FUNCTION_BLOCK "STD_LineSecStdSub2"	// FB 90
TITLE = Line and section control standard subroutines
//COPYRIGHT:   (C) 2004 BY  BUHLER LTD.
//                          CH-9240 UZWIL  SWITZERLAND
//
//PRODUCT:      STD_MU664    
//
//TITLE:        Line and section control standard subroutines
//              
//              Standardfunktionen für Linien und Sektionen              
//              
//
//--------------------------------------------------------------------------------
//
//IDENT:        AUTOR:              DEPT:                              DATE:
//STD_FB90.4.2  Ph. Engler          MU664                              27-Oct-2005
//              Sub2001: CmdStepOff modifyed
//STD_FB90.4.1  Ph. Engler          MU664                              22-Oct-2004
//              Sub2002: Extended section commands
//STD_FB90.4.0  Ph. Engler          MU664                              02-Sep-2004
//              Sub1055: StaDPFault as SubCode
//              Sub2055: StaDPFault as SubCode
//STD_FB90.3.4  Ph. Engler          MU664                              02-Jul-2004
//              Sub2003: No immediate stop anymore, its done from FC60 Move data
//STD_FB90.3.3  Ph. Engler          MU664                              23-Jun-2004
//              Sub1061/1062: BEA added
//STD_FB90.3.2  Ph. Engler          MU664                              02-Apr-2004
//              Sub2071: SectionState integrated   
//STD_FB90.3.1  Ph. Engler          MU664                              25-Mar-2004
//              Sub1061: Fault corrected, wrong tmp
//STD_FB90.3.0  Ph. Engler          MU664                              19-Feb-2004
//              Sub1061: General group info code for 64 objects
//STD_FB90.2.6  Ph. Engler          MU664                              12-Feb-2004
//              Sub1062: Maintenance info code
//STD_FB90.2.5  Ph. Engler          MU664                              28-Aug-2003
//              Sub1055: Handling of feeding section
//STD_FB90.2.4  Ph. Engler          MU664                              04-Aug-2003
//              Sub1061: Use LC to handle tmpLin_GenGrpCoulorCode
//STD_FB90.2.3  Ph. Engler          MU664                              29-Jul-2003
//              Sub1061: InOutValue3 stored to tmpDInt
//STD_FB90.2.2  Ph. Engler          MU664                              21-Jun-2003
//              Sub1051 corrected, yellow and blue
//STD_FB90.2.1  A.Egli              CT3                                14-Mai-2003
//              Sub1001: On Off Command Line
//STD_FB90.2.0  A.Egli              CT3                                18-Oct-2002
//              New release: Function moved from FC120 to FB90
//STD_FC120.1.12Ph. Engler          MU664                              23-Aug-2002
//              - Function (4,1) added: Search group manual mode
//STD_FC120.1.11Ph. Engler          MU664                              30-Apr-2002
//              - Function (1,55) and (2,55) modified: Stopping/Stopped
//STD_FC120.1.10Ph. Engler          MU664                              21-Mar-2002
//              - Function (2,55): starting until S.ToSSW.infStarted
//STD_FC120.1.9 Ph. Engler          MU664                              12-Mar-2002
//              Status codes for WinCoS implemented:
//              - General group colour code
//              - Line and Section info code
//STD_FC120.1.8 Ph. Engler          MU664                              20-Mar-2001
//              Line status colour for 2-4 section implemented
//STD_FC120.1.7 Ph. Engler          MU664                              20-Dec-2000
//              Pre stop weight for cmdSequenceStop
//STD_FC120.1.6 Ph. Engler          MU664                              14-Dec-2000
//              - Substitude Bincode into recipe extended, InCode 3 
//              - JS Job paramter flags (2,2) Sta-Address corrected
//STD_FC120.1.5 Ph. Engler          MU664                              01-Nov-2000
//              CmdSequenceStop only if section is in StActive           
//STD_FC120.1.4 Ph. Engler          MU664                              19-Okt-2000
//              Update SND-Binlist staSameSndRcv:
//               Suppression of the error meassage 'bin not found'
//STD_FC120.1.3 Ph. Engler          MU664                              28-Jun-2000
//              Section text and colour code extension 
//              with code 702, 703 and 1402
//STD_FC120.1.2 Ph. Engler          MU664                              04-May-2000
//              LS Line state/fault protocolling (1,10)
//               esXXX corrected 
//STD_FC120.1.1 Ph. Engler          MU664                              29-Mar-2000
//              Line log messages implemented
//STD_FC120.1.0 Ph. Engler          MU664                              05-Jan-2000
//              1st Release
//
//--------------------------------------------------------------------------------
//
//PURPOSE:      
//
//RESTRICTIONS:
//
//--------------------------------------------------------------------------------
//
AUTHOR : PE
FAMILY : STD
VERSION : 4.1
VAR_INPUT
  InCode : INT ;
END_VAR
VAR
  Para : STRUCT
   ParSecNr : INT  := 1;
   ParLineDB_ParFirstSecDB : INT  := 320;
   spare4 : INT ;
   ParNextSecDB : INT ;	//Next section DB of this project line
   ParSecDataFirstByte : INT  := 240;
   ParSecDataLenNomValue : INT  := 20;
   ParSecDataLenAcValue : INT  := 20;
   ParBinDataFirstByte : INT  := 300;
   ParBinDataLength : INT  := 72;
  END_STRUCT ;
  VarTemp : STRUCT
   InOutValue1 : INT ;
   InOutValue2 : INT ;
   InOutValue3 : DINT ;
   InOutValue4 : DINT ;
   InOutValue5 : DINT ;
   InOutValue6 : DINT ;
  END_STRUCT ;
  ChangeBit : STRUCT
   spare : BYTE ;
   CBit1 : BOOL ;
   CBit2 : BOOL ;
   CBit3 : BOOL ;
   CBit4 : BOOL ;
  END_STRUCT ;
  ToASW : STRUCT
   spare00 : WORD ;
   CmdModify : BOOL ;
   CmdNewBatch : BOOL ;
   CmdDataMoved : BOOL ;
   InfSameJobPrevSec : BOOL ;
   InfSameJobNextSec : BOOL ;
   InfSameBatchPrevSec : BOOL ;
   InfSameBatchNextSec : BOOL ;
   InfSameJobLineDB : BOOL ;	//Job in reveive box is equal
   InfEmptyingTimeEnd : BOOL ;
   InfWayAdjustTimeEnd : BOOL ;
   spare32 : BOOL ;
   spare33 : BOOL ;
   spare34 : BOOL ;
   spare35 : BOOL ;
   spare36 : BOOL ;
   InfDataReady : BOOL ;
   Func : UDT 10601;
   Transition : STRUCT
    spare00 : BYTE ;
    ToPassive : BOOL ;
    ToWait : BOOL ;
    ToActive : BOOL ;
    ToReady : BOOL ;
    ToEmptying : BOOL ;
    ToEmptied : BOOL ;
    ToIdling : BOOL ;
   END_STRUCT ;
   spare10 : WORD ;
   spare12 : DWORD ;
   spare16 : DWORD ;
  END_STRUCT ;
  ToSSW : STRUCT
   InfStopped : BOOL ;
   spare01 : BOOL ;
   InfStarted : BOOL ;
   spare03 : BOOL ;
   spare04 : BOOL ;
   InfFeeding : BOOL ;
   spare06 : BOOL ;
   spare07 : BOOL ;
   spare00 : BOOL ;
   CmdGotoActive : BOOL ;
   CmdGotoReady : BOOL ;
   CmdGotoEmptying : BOOL ;
   CmdGotoEmptied : BOOL ;
   CmdGotoIdling : BOOL ;
   CmdGotoPassive : BOOL ;
   spare17 : BOOL ;
   InfReadyForNewBatch : BOOL ;
   CmdSendResult : BOOL ;
   InfPulseTimer : BOOL ;
   CmdNewWay : BOOL ;
   spare24 : BOOL ;
   spare25 : BOOL ;
   spare26 : BOOL ;
   InfReleaseEmptyingTime : BOOL ;
   Func : UDT 10601;
   InPrevSecDB : INT ;	//Previouse section DB in product flow
   InNextSecDB : INT ;	//Next section DB in product flow
   spare12 : DWORD ;
   spare16 : DWORD ;
  END_STRUCT ;
  PCWrite : STRUCT 	//PC Write : Section Data
   Hsk : STRUCT
    Q_Status : BOOL ;
    Q_Result : BOOL ;
    spare02 : BOOL ;
    spare03 : BOOL ;
    spare04 : BOOL ;
    spare05 : BOOL ;
    Q_MDEEData : BOOL ;	//Acknowledge data sended to MDEE by PCC
    Q_MYRAData : BOOL ;	//Acknowledge data sended to MYRA by PCC
    F_Define : BOOL ;
   END_STRUCT ;
   spare2 : WORD ;
   Func : UDT 10601;
   Value1 : INT ;
   Value2 : INT ;
   Value3 : INT ;
   ParWayAdjustTime : INT  := 2;
   Value5 : INT ;
   ParEmptyingTime : INT  := 20;
  END_STRUCT ;
  PCRead : STRUCT 	//PC Read : Section Data
   Hsk : STRUCT
    F_Status : BOOL ;
    F_Result : BOOL ;
    F_2 : BOOL ;
    F_3 : BOOL ;
    F_4 : BOOL ;
    F_5 : BOOL ;
    F_MDEEData : BOOL ;	//Request PCC to send data to MDEE
    F_MYRAData : BOOL ;	//Request PCC to send data to MYRA
   END_STRUCT ;
   ErrElement : INT ;
   ErrCode : INT ;
   ErrObject : INT ;	//(*new*)
   Step : STRUCT
    spare : BYTE ;
    StPassive : BOOL ;
    StWait : BOOL ;
    StActive : BOOL ;
    StReady : BOOL ;	//Line= Idling
    StEmptying : BOOL ;
    StEmptied : BOOL ;
    StIdling : BOOL ;
   END_STRUCT ;
   State : STRUCT
    spare : BYTE ;
    StStopped : BOOL ;
    StStarting : BOOL ;
    StStarted : BOOL ;
    StStopping : BOOL ;
    spare04 : BOOL ;
    StFeeding : BOOL ;
   END_STRUCT ;
   Fault : UDT 10602;
   Status : UDT 10603;
   InfoCode : INT ;
   SectionState : INT ;	//Line: GenGrpColorCode
   ExtStatus : INT ;
   OutWayAdjustTime_ExtOn : INT ;
   OutStartWarningTime : INT ;	//Copy of Startwarning modul
   OutEmptyingTime : INT ;
   Value7 : INT ;
   Value8 : INT ;
   Value9 : INT ;
   Value10 : INT ;
   Value11 : INT ;
   Value12 : INT ;
   Value13 : INT ;
   Value14 : INT ;
   Value15 : INT ;
   Value16 : INT ;
   Value17 : INT ;
   ExtFuncOn : INT ;
   Value19 : INT ;
  END_STRUCT ;
  JobNom : STRUCT 	//PC Read: Job header: Nominal values
   JobNr : DINT ;
   JobWeight : DINT ;	//Total Job weight
   BatchNo : INT  := 10;	//Number of batch requested form PC
   ScaleUsed : ARRAY  [1 .. 64 ] OF BOOL ;
   RecipeNr : INT ;
   BatchWeight : DINT ;
   BatchMinPpm : INT ;	//Minimum batch size [0.1%]
   BatchMaxPpm : INT ;	//Maximum batch size [0.1%]
   BatchNoOffset : INT ;	//Batch number of first batch
   MixingTime : INT ;	//Mixing time
   JobChangeTime : INT ;	//Job change time
   FeedingTime : INT ;	//Feeding Time
   Value13 : INT ;
   Value14 : INT ;
  END_STRUCT ;
  JobAc : STRUCT 	//PC Read: Job header: Actual values
   StaBatch : STRUCT
    spare0 : BOOL ;
    spare1 : BOOL ;
    spare2 : BOOL ;
    spare3 : BOOL ;
    spare4 : BOOL ;
    spare5 : BOOL ;
    StaEmptyingBatch : BOOL ;
    StaScaleRecipeValid : BOOL ;
    StaErrBatch : BOOL ;
    StaHandAddReady : BOOL ;
    StaRegistrated : BOOL ;
    StaLastBatch : BOOL ;
    StaDone : BOOL ;
   END_STRUCT ;
   JobWeight : DINT ;
   BatchNo : INT ;
   BatchNoCal : INT ;
   BatchWeightTarget : DINT ;	//Calculated target batch weight
   BatchWeightActual : DINT ;	//Actual weight of all dosed ingredient
   BatchSizePpm : INT ;	//Calculated batch size [1/1000]
   BatchValue8 : INT ;
   BatchValue9 : INT ;
   MixingTime : INT ;	//Mixing time
   JobChangeTime : INT ;	//Job change time
   FeedingTime : INT ;	//Feeding Time
   RecipePlace : INT ;	//Actual recipe place
   Value16 : INT ;
   Value17 : INT ;
   Value18 : INT ;
   Value19 : INT ;
  END_STRUCT ;
END_VAR
VAR_TEMP
  TmpWord : WORD ;
  TmpInt : INT ;
  TmpDInt : DINT ;
  TmpBool : BOOL ;
  tmpLineStStopped : BOOL ;
  tmpLineStaAutostart : BOOL ;
  tmpLineInfFeeding : BOOL ;
  DB9SecArray : DWORD ;	//Address Pointer Section in DB9
  tmpSecDB : INT ;
  tmpAddrGrInterfaceSec : DINT ;	//Pointer to Interface in section DB
  tmpLineDB : INT ;
  tmpRelevantGroups32_1 : DINT ;
  tmpSec_GenGrpCoulorCode : STRUCT
   lightGrey : BOOL ;
   Bit1 : BOOL ;
   darkGreen : BOOL ;
   magenta : BOOL ;
   red : BOOL ;
  END_STRUCT ;
  tmpLin_GenGrpCoulorCode : STRUCT
   lightGrey : BOOL ;
   Bit1 : BOOL ;
   darkGreen : BOOL ;
   magenta : BOOL ;
   red : BOOL ;
  END_STRUCT ;
  tmpStateColorS1 : STRUCT
   white : BOOL ;
   yellow : BOOL ;
   blue : BOOL ;
   dark_green : BOOL ;
   green : BOOL ;
   light_green : BOOL ;
   mangenta : BOOL ;
   red : BOOL ;
   Bit8 : BOOL ;
   Bit9 : BOOL ;
   Bit10 : BOOL ;
   Bit11 : BOOL ;
   Bit12 : BOOL ;
   brown : BOOL ;
   orange : BOOL ;
   tuerkis : BOOL ;
  END_STRUCT ;
  tmpStateColorS2 : STRUCT
   white : BOOL ;
   yellow : BOOL ;
   blue : BOOL ;
   dark_green : BOOL ;
   green : BOOL ;
   light_green : BOOL ;
   mangenta : BOOL ;
   red : BOOL ;
   Bit8 : BOOL ;
   Bit9 : BOOL ;
   Bit10 : BOOL ;
   Bit11 : BOOL ;
   Bit12 : BOOL ;
   brown : BOOL ;
   orange : BOOL ;
   tuerkis : BOOL ;
  END_STRUCT ;
  tmpStateColorS3 : STRUCT
   white : BOOL ;
   yellow : BOOL ;
   blue : BOOL ;
   dark_green : BOOL ;
   green : BOOL ;
   light_green : BOOL ;
   mangenta : BOOL ;
   red : BOOL ;
   Bit8 : BOOL ;
   Bit9 : BOOL ;
   Bit10 : BOOL ;
   Bit11 : BOOL ;
   Bit12 : BOOL ;
   brown : BOOL ;
   orange : BOOL ;
   tuerkis : BOOL ;
  END_STRUCT ;
  tmpStateColorS4 : STRUCT
   white : BOOL ;
   yellow : BOOL ;
   blue : BOOL ;
   dark_green : BOOL ;
   green : BOOL ;
   light_green : BOOL ;
   mangenta : BOOL ;
   red : BOOL ;
   Bit8 : BOOL ;
   Bit9 : BOOL ;
   Bit10 : BOOL ;
   Bit11 : BOOL ;
   Bit12 : BOOL ;
   brown : BOOL ;
   orange : BOOL ;
   tuerkis : BOOL ;
  END_STRUCT ;
  tmpStateColorLine : STRUCT
   white : BOOL ;
   yellow : BOOL ;
   blue : BOOL ;
   dark_green : BOOL ;
   green : BOOL ;
   light_green : BOOL ;
   mangenta : BOOL ;
   red : BOOL ;
   Bit8 : BOOL ;
   Bit9 : BOOL ;
   Bit10 : BOOL ;
   Bit11 : BOOL ;
   Bit12 : BOOL ;
   brown : BOOL ;
   orange : BOOL ;
   tuerkis : BOOL ;
  END_STRUCT ;
  tmpInCode : INT ;
  tmpNoOfSec : INT ;
  tmpInfFeedingSection : INT ;
  tmpDInt2 : DINT ;
  tmpRelevantGroups64_33 : DINT ;
  tmpUserState : STRUCT
   stEmptying : BOOL ;
   stEmptied : BOOL ;
   stIdling : BOOL ;
   stFault : BOOL ;
   stHand : BOOL ;
   stHold : BOOL ;
   stStep : BOOL ;
   spare : BOOL ;
   stPassive : BOOL ;
   stWait : BOOL ;
   stStarting : BOOL ;
   stStarted : BOOL ;
   stStopping : BOOL ;
   stStopped : BOOL ;
   stFeeding : BOOL ;
   stReady : BOOL ;
  END_STRUCT ;
END_VAR
BEGIN
NETWORK
TITLE = Init
      LAR2  P##InCode;
      L     DINO;
      T     #tmpLineDB;
      T     #tmpSecDB;
// 
      L     #InCode;
      T     #tmpInCode;	// Use only this tag within the procedures
NETWORK
TITLE = Sub1001: LS Line On Off Command
//Called by line controler subroutines, with opened L-DB
      L     #InCode;
      L     1001;
      <>I;
      JC    LS01;
      L     #PCWrite.Value1;	// PCWrite.ExtFuncOn 
      T     #PCRead.OutWayAdjustTime_ExtOn;
//-Update ExtStatus------------------------
      L     #PCRead.ExtStatus;	// ExtStatus
      L     #PCWrite.Value1;	// PCWrite.ExtFuncOn 
      OD;	// 
      L     #PCWrite.Value2;	// PCWrite.ExtFuncOff 
      INVD;	//  
      AD;	//  
      T     #PCRead.ExtStatus;	//->ExtStatus
//Reset on commands 
      L     0;
      T     #PCWrite.Value1;	// PCWrite.ExtFuncOn 
//Reset off commands 
      L     0;
      T     #PCWrite.Value2;	// PCWrite.ExtFuncOff 
      BEU;
LS01: NOP   0;
NETWORK
TITLE = Sub1010: LS Line state/fault protocolling
//Called by line controler subroutines, with opened L-DB
//
//Output: LineDB.VarTemp.InOutValue1 = LineMsg
      L     #InCode;
      L     1010;
      <>I;
      JC    LS00;
//-Init var---
      L     0;
      T     MW 2018;
//Read old value: PCRead.StateColor
      L     #PCRead.InfoCode;
      LAR1  P##tmpStateColorS1;	// LineDB.PCRead.StateColor
      T     LW [AR1,P#0.0];	//-->tmpStateColorS1
//-Generate summary step---
      A     #tmpStateColorS1.tuerkis;	// 
      =     M 2019.3;	// --> LineMsg.suspended
      SET;
      S     M 2019.0;	// --> LineMsg.terminated
      S     M 2019.1;	// --> LineMsg.stopped
      R     M 2019.2;	// --> LineMsg.started
      R     M 2019.4;	// --> LineMsg.faulted
      R     M 2019.5;	// --> LineMsg.warning
      R     M 2018.0;	// --> LineMsg.SenderEmpty
      R     M 2018.3;	// --> LineMsg.allPreselectRcvFull
      R     M 2018.4;	// --> LineMsg.MachinesNotAvailable
      L     #Para.ParLineDB_ParFirstSecDB;	// Para.ParFirstSecDB   
LOOP: T     #tmpSecDB;
      OPN   DI [#tmpSecDB];
      AN    #PCRead.Step.StPassive;	// Section
      AN    #PCRead.Step.StIdling;	// Section
      R     M 2019.0;	// --> LineMsg.terminated
      AN    #PCRead.State.StStopped;	// Section
      ON    #PCRead.Status.StaImmediateStopASW;	// Section
      R     M 2019.1;	// --> LineMsg.stopped
      AN    #PCRead.Step.StPassive;	// Section
      AN    #PCRead.Step.StIdling;	// Section
      S     M 2019.2;	// --> LineMsg.started
      A     #PCRead.Fault.EsMech;	// Section
      AN    #PCRead.Step.StPassive;	// Section
      AN    #PCRead.Step.StIdling;	// Section
      S     M 2019.4;	// --> LineMsg.faulted
      A     #PCRead.Fault.EsWarning;	// Section
      AN    #PCRead.Step.StPassive;	// Section
      AN    #PCRead.Step.StIdling;	// Section
      S     M 2019.5;	// --> LineMsg.warning
      A     #PCRead.Fault.EsEmpty;	// Section
      AN    #PCRead.Step.StPassive;	// Section
      AN    #PCRead.Step.StIdling;	// Section
      S     M 2018.0;	// --> LineMsg.SenderEmpty
      A     #PCRead.Fault.EsFull;	// Section
      AN    #PCRead.Step.StPassive;	// Section
      AN    #PCRead.Step.StIdling;	// Section
      S     M 2018.3;	// --> LineMsg.allPreselectRcvFull
      A     #PCRead.Fault.EsWayConflict;	// Section
      AN    #PCRead.Step.StPassive;	// Section
      AN    #PCRead.Step.StIdling;	// Section
      S     M 2018.4;	// --> LineMsg.MachinesNotAvailable
//-Check next section---
      L     0;
      L     #Para.ParNextSecDB;	// Section
      <>I;
      JC    LOOP;
//-Return messages---
      OPN   DI [#tmpLineDB];
      L     MW 2018;	// LineMsg
      T     #VarTemp.InOutValue1;
      BEU;
LS00: NOP   0;
NETWORK
TITLE = Sub1051: C1 Line status colour for 1 section
//Called by line controler subroutines
      L     #InCode;
      L     1051;
      <>I;
      JC    C100;
//Init
      L     0;
      LAR1  P##tmpStateColorLine;
      T     LW [AR1,P#0.0];	//-->tmpStateColorLine
//Read state of section 1
      L     #Para.ParLineDB_ParFirstSecDB;
      T     #tmpSecDB;
      OPN   DI [#tmpSecDB];	// Call 1st section
      L     #PCRead.InfoCode;	// Section
      LAR1  P##tmpStateColorS1;
      T     LW [AR1,P#0.0];	//-->tmpStateColorS1
//-Red----------------------------------
      A     #tmpStateColorS1.red;	// Section
      S     #tmpStateColorLine.red;
      JC    C101;
//-Magenta------------------------------
      A     #tmpStateColorS1.mangenta;	// Section
      S     #tmpStateColorLine.mangenta;
      JC    C101;
//-Turkis-------------------------------
      A     #tmpStateColorS1.tuerkis;	// Section
      S     #tmpStateColorLine.tuerkis;
      JC    C101;
//-Brown--------------------------------
      A     #tmpStateColorS1.brown;	// Section
      S     #tmpStateColorLine.brown;
      JC    C101;
//-Orange-------------------------------
      A     #tmpStateColorS1.orange;	// Section
      S     #tmpStateColorLine.orange;
      JC    C101;
//-Lightgreen---------------------------
      A     #tmpStateColorS1.light_green;	// Section
      S     #tmpStateColorLine.light_green;
      JC    C101;
//-Green--------------------------------
      A     #tmpStateColorS1.green;	// Section
      S     #tmpStateColorLine.green;
      JC    C101;
//-Darkgreen----------------------------
      A     #tmpStateColorS1.dark_green;	// Section
      S     #tmpStateColorLine.dark_green;
      JC    C101;
//-Yellow-------------------------------
      A     #tmpStateColorS1.yellow;	// Section
      S     #tmpStateColorLine.yellow;
      JC    C101;
//-Blue---------------------------------
      A     #tmpStateColorS1.blue;	// Section
      S     #tmpStateColorLine.blue;
      JC    C101;
//-White--------------------------------
      A     #tmpStateColorS1.white;	// Section
      S     #tmpStateColorLine.white;	//(default)
//-Data to PCC--------------------------
C101: OPN   DI [#tmpLineDB];
      LAR1  P##tmpStateColorLine;
      L     LW [AR1,P#0.0];	// tmpStateColorLine
      L     #PCRead.InfoCode;	// LineDB
      ==I;	// 
      BEC;
      S     #ChangeBit.CBit1;	// LineDB
      TAK;
      T     #PCRead.InfoCode;	// LineDB
      BEU;
C100: NOP   0;
NETWORK
TITLE = Sub1052: C2 Line status colour for 2 section
//Called by line controler subroutines
//
//Inputs :
// no
//Outputs:
// no
//
      L     #InCode;
      L     1052;
      <>I;
      JC    C200;
//Init
      L     0;
      LAR1  P##tmpStateColorLine;
      T     LW [AR1,P#0.0];	//-->tmpStateColorLine
//Read Status Section 1
      L     #Para.ParLineDB_ParFirstSecDB;
      T     #tmpSecDB;
      OPN   DI [#tmpSecDB];	// Call 1st section DB Para.ParFirstSecDB
      L     #PCRead.InfoCode;	// Section
      LAR1  P##tmpStateColorS1;
      T     LW [AR1,P#0.0];	//-->tmpStateColorS1
//Read Status Section2
      L     #Para.ParNextSecDB;	// Section
      T     #tmpSecDB;
      OPN   DI [#tmpSecDB];	// Call next section DB Para.ParNextSecDB
      L     #PCRead.InfoCode;	// Section
      LAR1  P##tmpStateColorS2;
      T     LW [AR1,P#0.0];	//-->tmpStateColorS2
      OPN   DI [#tmpLineDB];	// Call line DB .Para.ParLineDB
//-Red----------------------------------
      A     #tmpStateColorS1.red;
      O     #tmpStateColorS2.red;
      S     #tmpStateColorLine.red;
      JC    C201;
//-Magenta------------------------------
      A     #tmpStateColorS1.mangenta;
      O     #tmpStateColorS2.mangenta;
      S     #tmpStateColorLine.mangenta;
      JC    C201;
//-Turkis-------------------------------
      A     #tmpStateColorS1.tuerkis;
      O     #tmpStateColorS2.tuerkis;
      S     #tmpStateColorLine.tuerkis;
      JC    C201;
//-Brown--------------------------------
      A     #tmpStateColorS1.brown;
      O     #tmpStateColorS2.brown;
      S     #tmpStateColorLine.brown;
      JC    C201;
//-Orange-------------------------------
      A     #tmpStateColorS1.orange;
      O     #tmpStateColorS2.orange;
      S     #tmpStateColorLine.orange;
      JC    C201;
//-Lightgreen---------------------------
      A     #tmpStateColorS1.light_green;
      O     #tmpStateColorS2.light_green;
      S     #tmpStateColorLine.light_green;
      JC    C201;
//-Green--------------------------------
      A     #tmpStateColorS1.green;
      O     #tmpStateColorS2.green;
      S     #tmpStateColorLine.green;
      JC    C201;
//-Darkgreen----------------------------
      A     #tmpStateColorS1.dark_green;
      O     #tmpStateColorS2.dark_green;
      S     #tmpStateColorLine.dark_green;
      JC    C201;
//-Blue---------------------------------
      A     #tmpStateColorS1.blue;
      O     #tmpStateColorS2.blue;
      S     #tmpStateColorLine.blue;
      JC    C201;
//-Yellow-------------------------------
      A     #tmpStateColorS1.yellow;
      O     #tmpStateColorS2.yellow;
      S     #tmpStateColorLine.yellow;
      JC    C201;
//-White--------------------------------
      A     #tmpStateColorS1.white;
      A     #tmpStateColorS2.white;
      S     #tmpStateColorLine.white;	// (default)
//-Data to PCC--------------------------
C201: OPN   DI [#tmpLineDB];
      LAR1  P##tmpStateColorLine;
      L     LW [AR1,P#0.0];	// tmpStateColorLine
      L     #PCRead.InfoCode;	// LineDB
      ==I;
      BEC;
      S     #ChangeBit.CBit1;	// LineDB
      TAK;
      T     #PCRead.InfoCode;	// LineDB
      BEU;
C200: NOP   0;
NETWORK
TITLE = Sub1053: C3 Line status colour for 3 section
//Called by line controler subroutines
//
//Inputs :
// no
//Outputs:
// no
//
      L     #InCode;
      L     1053;
      <>I;
      JC    C300;
//Init
      L     0;
      LAR1  P##tmpStateColorLine;
      T     LW [AR1,P#0.0];	//-->tmpStateColorLine
//Read Status Section1
      L     #Para.ParLineDB_ParFirstSecDB;
      T     #tmpSecDB;
      OPN   DI [#tmpSecDB];	// Call 1st section DB Para.ParFirstSecDB
      L     #PCRead.InfoCode;	// Section
      LAR1  P##tmpStateColorS1;
      T     LW [AR1,P#0.0];	//-->tmpStateColorS1
//Read Status Section2
      L     #Para.ParNextSecDB;	// Section
      T     #tmpSecDB;
      OPN   DI [#tmpSecDB];	// Call next section DB Para.ParNextSecDB
      L     #PCRead.InfoCode;	// Section
      LAR1  P##tmpStateColorS2;
      T     LW [AR1,P#0.0];	//-->tmpStateColorS2
//Read Status Section3
      L     #Para.ParNextSecDB;	// Section
      T     #tmpSecDB;
      OPN   DI [#tmpSecDB];	// Call next section DB Para.ParNextSecDB
      L     #PCRead.InfoCode;	// Section
      LAR1  P##tmpStateColorS3;
      T     LW [AR1,P#0.0];	//-->tmpStateColorS3
//-Red----------------------------------
      OPN   DI [#tmpLineDB];
      A     #tmpStateColorS1.red;
      O     #tmpStateColorS2.red;
      O     #tmpStateColorS3.red;
      S     #tmpStateColorLine.red;
      JC    C301;
//-Magenta------------------------------
      A     #tmpStateColorS1.mangenta;
      O     #tmpStateColorS2.mangenta;
      O     #tmpStateColorS3.mangenta;
      S     #tmpStateColorLine.mangenta;
      JC    C301;
//-Turkis-------------------------------
      A     #tmpStateColorS1.tuerkis;
      O     #tmpStateColorS2.tuerkis;
      O     #tmpStateColorS3.tuerkis;
      S     #tmpStateColorLine.tuerkis;
      JC    C301;
//-Brown--------------------------------
      A     #tmpStateColorS1.brown;
      O     #tmpStateColorS2.brown;
      O     #tmpStateColorS3.brown;
      S     #tmpStateColorLine.brown;
      JC    C301;
//-Orange-------------------------------
      A     #tmpStateColorS1.orange;
      O     #tmpStateColorS2.orange;
      O     #tmpStateColorS3.orange;
      S     #tmpStateColorLine.orange;
      JC    C301;
//-Lightgreen---------------------------
      A     #tmpStateColorS1.light_green;
      O     #tmpStateColorS2.light_green;
      O     #tmpStateColorS3.light_green;
      S     #tmpStateColorLine.light_green;
      JC    C301;
//-Green--------------------------------
      A     #tmpStateColorS1.green;
      O     #tmpStateColorS2.green;
      O     #tmpStateColorS3.green;
      AN    #tmpStateColorS2.dark_green;
      S     #tmpStateColorLine.green;
      JC    C301;
//-Darkgreen----------------------------
//      U     #tmpStateColorS1.dark_green
      A     #tmpStateColorS2.dark_green;
//      U     #tmpStateColorS3.dark_green
      S     #tmpStateColorLine.dark_green;
      JC    C301;
//-Blue---------------------------------
      A     #tmpStateColorS1.blue;
      O     #tmpStateColorS2.blue;
      O     #tmpStateColorS3.blue;
      S     #tmpStateColorLine.blue;
      JC    C301;
//-Yellow-------------------------------
//      U     #tmpStateColorS1.yellow
      A     #tmpStateColorS2.yellow;
//      U     #tmpStateColorS3.yellow
      S     #tmpStateColorLine.yellow;
      JC    C301;
//-White--------------------------------
//      U     #tmpStateColorS1.white
      A     #tmpStateColorS2.white;
      A     #tmpStateColorS3.white;
      S     #tmpStateColorLine.white;	// (default)
      JC    C301;
//-Data to PCC--------------------------
C301: OPN   DI [#tmpLineDB];
      LAR1  P##tmpStateColorLine;
      L     LW [AR1,P#0.0];	// tmpStateColorLine
      L     #PCRead.InfoCode;	// LineDB
      ==I;	// 
      BEC;
      S     #ChangeBit.CBit1;	// LineDB
      TAK;
      T     #PCRead.InfoCode;	// LineDB
      BEU;
C300: NOP   0;
NETWORK
TITLE = Sub1054: C4 Line status colour for 4 section
//Called by line controler subroutines
      L     #InCode;
      L     1054;
      <>I;
      JC    C400;
//Init
      L     0;
      LAR1  P##tmpStateColorLine;
      T     LW [AR1,P#0.0];	//-->tmpStateColorLine
//Read Status Section1
      L     #Para.ParLineDB_ParFirstSecDB;
      T     #tmpSecDB;
      OPN   DI [#tmpSecDB];	// Call 1st section DB Para.ParFirstSecDB
      L     #PCRead.InfoCode;	// Section
      LAR1  P##tmpStateColorS1;
      T     LW [AR1,P#0.0];	//-->tmpStateColorS1
//Read Status Section2
      L     #Para.ParNextSecDB;	// Section
      T     #tmpSecDB;
      OPN   DI [#tmpSecDB];	// Call next section DB Para.ParNextSecDB
      L     #PCRead.InfoCode;	// Section
      LAR1  P##tmpStateColorS2;
      T     LW [AR1,P#0.0];	//-->tmpStateColorS2
//Read Status Section3
      L     #Para.ParNextSecDB;	// Section
      T     #tmpSecDB;
      OPN   DI [#tmpSecDB];	// Call next section DB Para.ParNextSecDB
      L     #PCRead.InfoCode;	// Section
      LAR1  P##tmpStateColorS3;
      T     LW [AR1,P#0.0];	//-->tmpStateColorS3
//Read Status Section4
      L     #Para.ParNextSecDB;	// Section
      T     #tmpSecDB;
      OPN   DI [#tmpSecDB];	// Call next section DB Para.ParNextSecDB
      L     #PCRead.InfoCode;	// Section
      LAR1  P##tmpStateColorS4;
      T     LW [AR1,P#0.0];	//-->tmpStateColorS4
      OPN   DI [#tmpLineDB];	// Call line DB 
// 
//-Red----------------------------------
      A     #tmpStateColorS1.red;
      O     #tmpStateColorS2.red;
      O     #tmpStateColorS3.red;
      O     #tmpStateColorS4.red;
      S     #tmpStateColorLine.red;
      JC    C401;
//-Magenta------------------------------
      A     #tmpStateColorS1.mangenta;
      O     #tmpStateColorS2.mangenta;
      O     #tmpStateColorS3.mangenta;
      O     #tmpStateColorS4.mangenta;
      S     #tmpStateColorLine.mangenta;
      JC    C401;
//-Turkis-------------------------------
      A     #tmpStateColorS1.tuerkis;
      O     #tmpStateColorS2.tuerkis;
      O     #tmpStateColorS3.tuerkis;
      O     #tmpStateColorS4.tuerkis;
      S     #tmpStateColorLine.tuerkis;
      JC    C401;
//-Yellow-------------------------------
      A     #tmpStateColorS1.yellow;
      A     #tmpStateColorS2.yellow;
      A     #tmpStateColorS3.yellow;
      A     #tmpStateColorS4.yellow;
      S     #tmpStateColorLine.yellow;
      JC    C401;
//-Brown--------------------------------
      A     #tmpStateColorS1.brown;
      O     #tmpStateColorS2.brown;
      O     #tmpStateColorS3.brown;
      O     #tmpStateColorS4.brown;
      S     #tmpStateColorLine.brown;
      JC    C401;
//-Orange-------------------------------
      A     #tmpStateColorS1.orange;
      O     #tmpStateColorS2.orange;
      O     #tmpStateColorS3.orange;
      O     #tmpStateColorS4.orange;
      S     #tmpStateColorLine.orange;
      JC    C401;
//-Lightgreen---------------------------
//      U     #tmpStateColorS1.light_green
//      U     #tmpStateColorS2.light_green
//      U     #tmpStateColorS3.light_green
//      U     #tmpStateColorS4.light_green
      CLR;
      S     #tmpStateColorLine.light_green;
      JC    C401;
//-Green--------------------------------
//      U     #tmpStateColorS1.green
//      U     #tmpStateColorS2.green
//      U     #tmpStateColorS3.green
//      U     #tmpStateColorS4.green
      CLR;
      S     #tmpStateColorLine.green;
      JC    C401;
//-Blue---------------------------------
      A     #tmpStateColorS1.white;
      A     #tmpStateColorS2.white;
      A     #tmpStateColorS3.white;
      A     #tmpStateColorS4.blue;
      S     #tmpStateColorLine.blue;
      JC    C401;
//-Darkgreen----------------------------
//      U     #tmpStateColorS1.dark_green
//      U     #tmpStateColorS2.dark_green
//      U     #tmpStateColorS3.dark_green
//      U     #tmpStateColorS4.dark_green
      A     #PCRead.Step.StActive;	// LineDB 
      O     #PCRead.Step.StReady;	// LineDB 
      S     #tmpStateColorLine.dark_green;
      JC    C401;
//-White--------------------------------
//      U     #tmpStateColorS1.white
//      U     #tmpStateColorS2.white
//      U     #tmpStateColorS3.white
//      U     #tmpStateColorS4.white
      A     #PCRead.Step.StPassive;	// LineDB
      O     #PCRead.Step.StIdling;	// LineDB
      S     #tmpStateColorLine.white;	// (default)
      JC    C401;
//-Data to PCC--------------------------
C401: OPN   DI [#tmpLineDB];
      LAR1  P##tmpStateColorLine;
      L     LW [AR1,P#0.0];	// tmpStateColorLine
      L     #PCRead.InfoCode;	// LineDB
      ==I;	// 
      BEC;
      S     #ChangeBit.CBit1;	// LineDB
      TAK;
      T     #PCRead.InfoCode;	// LineDB
      BEU;
C400: NOP   0;
NETWORK
TITLE = Sub1055: I1 Line info code for x sections WinCoS
      L     #InCode;
      L     1055;
      <>I;
      A(;	//[2.5]
      L     #InCode;	//[2.5]
      L     1155;	//[2.5]
      <>I;	//[2.5]
      );	//[2.5]
      A(;	//[2.5]
      L     #InCode;	//[2.5]
      L     1255;	//[2.5]
      <>I;	//[2.5]
      );	//[2.5]
      JC    I100;
// 
//-Begin-Scan all sections---
      L     #InCode;	//[2.5]
      L     1055;	//[2.5]
      -I;	//[2.5]
      L     100;	//[2.5]
      /I;	//[2.5]
      T     #tmpInfFeedingSection;	//[2.5]
      L     1;	//[2.5]
      T     #tmpNoOfSec;	//[2.5]
      L     #Para.ParLineDB_ParFirstSecDB;	// LineDB
      T     #tmpSecDB;
      OPN   DI [#tmpSecDB];	// Call Section DB
      SET;
      =     #tmpLineStaAutostart;
      =     #tmpLineStStopped;
      =     #tmpLineInfFeeding;
I1L1: AN    #PCRead.Status.StaAutostart;	// Section
      R     #tmpLineStaAutostart;
      AN    #PCRead.State.StStopped;	// Section
      AN    #PCRead.State.StStopping;	// Section
      R     #tmpLineStStopped;
      A(;	//[2.5]
      L     #tmpNoOfSec;	//[2.5]
      L     #tmpInfFeedingSection;	//[2.5]
      ==I;	//[2.5]
      O(;	//[2.5]
      L     #tmpInfFeedingSection;	//[2.5]
      L     0;	//[2.5]
      ==I;	//[2.5]
      );	//[2.5]
      );	//[2.5]
      AN    #ToSSW.InfFeeding;	// Section
      R     #tmpLineInfFeeding;
//-End-Scan all sections--- 
      L     #tmpNoOfSec;	//[2.5]
      +     1;	//[2.5]
      T     #tmpNoOfSec;	//[2.5]
      L     #Para.ParNextSecDB;	// Section
      L     0;
      <>I;
      JCN   I101;
      L     #Para.ParNextSecDB;
      T     #tmpSecDB;
      OPN   DI [#tmpSecDB];	// Call next S-DB
      JU    I1L1;
//-End-Scan all sections---
//===Line =============================================================
I101: OPN   DI [#tmpLineDB];	// Call L-DB
//=Build MainInfoCode=================
//-Fault------------------------------
      A     #PCRead.Fault.EsMech;	// LineDB
      O     #PCRead.Fault.EsDosing;	// LineDB
      O     #PCRead.Fault.EsBatchSize;	// LineDB
      O     #PCRead.Fault.EsRefillLevel;	// LineDB
      AN    #PCRead.Step.StPassive;	// LineDB
      AN    #PCRead.Step.StIdling;	// LineDB
      L     2#100000000000000;	// bit_main_status.passiv
      L     1500;	// code.Fault
      JC    I102;
//-Passive------------------------------
      A     #PCRead.Step.StPassive;	// LineDB
      L     2#1;	// bit_main_status.passiv
      L     100;	// code.st_passiv
      JC    I102;
//-AvailableTest------------------------
      A     #PCRead.Step.StActive;	// LineDB
      O     #PCRead.Step.StReady;	// LineDB
      A     #PCRead.Fault.EsWayConflict;	// LineDB
      L     2#100;	// bit_main_status.AvailableTest 
      L     300;	// code.st_AvailableTest
      JC    I102;
//-Stopped------------------------------
      A     #PCRead.Step.StActive;	// LineDB
      O     #PCRead.Step.StReady;	// LineDB
      A     #tmpLineStStopped;
      L     2#10000000000000;	// bit_main_status.stopped 
      L     1400;	// code.st_stopped
      JC    I102;
//-Suspended----------------------------
      A     #PCRead.Step.StActive;	// LineDB
      O     #PCRead.Step.StReady;	// LineDB
      AN    #tmpLineInfFeeding;
      L     2#100000;	// bit_main_status.suspended 
      L     600;	// code.st_suspended
      JC    I102;
//-Running------------------------------
      A     #PCRead.Step.StActive;	// LineDB
      O     #PCRead.Step.StReady;	// LineDB
      L     2#1000000;	// bit_main_status.running 
      L     700;	// code.st_running
      JC    I102;
//-Idling-------------------------------
      A     #PCRead.Step.StIdling;	// LineDB
      L     2#100000000000;	// bit_main_status.idling 
      L     1200;	// code.st_idling
      JC    I102;
//-No State-----------------------------
      L     2#0;	// bit_main_status.no_state 
      L     0;	// code.st_no_state
I102: T     #TmpInt;	// line text status
      TAK;
      T     #TmpWord;	// bit_main_status
// 
//=Build SubInfoCode====================
//-Fault--------------------------------
      OPN   DI [#tmpLineDB];
//-DPFault------------------------------
      L     #TmpWord;	// bit_main_status
      L     2#111111111111111;	// mask with restart code
      AW;
      JZ    I1N1;
      A     #PCRead.Status.StaDPFault;	// LineDB
      L     7;	// code.dpfault
      JC    I103;
//-ReStart------------------------------
I1N1: L     #TmpWord;	// bit_main_status
      L     2#110000001100000;	// mask with restart code
      AW;
      JZ    I1N2;
      A     #PCRead.Status.StaImmediateStop;	// LineDB
      O     #PCRead.Status.StaTransferOff;	// LineDB
      O     #PCRead.Status.StaFeedOff;	// LineDB
      AN    #PCRead.Status.StaStep;	// LineDB
      ON    #tmpLineStaAutostart;
      L     3;	// code.restart
      JC    I103;
//-Step mode----------------------------
I1N2: L     #TmpWord;	// bit_main_status
      L     2#110000001101101;	// mask with step-mode code
      AW;
      JZ    I1N3;
      A     #PCRead.Status.StaStep;	// LineDB
      L     4;	// code.Step-mode
      JC    I103;
//-Hold---------------------------------
I1N3: L     #TmpWord;	// bit_main_status
      L     2#110100001101101;	// mask with step-mode code
      AW;
      JZ    I1N4;
      A     #PCRead.Status.StaHold;	// LineDB
      L     6;	// code.Step-mode
      JC    I103;
//-Warning------------------------------
I1N4: L     #TmpWord;	// bit_main_status
      L     2#110100001101000;	// mask with warning code
      AW;
      JZ    I1N5;
      A     #PCRead.Fault.EsWarning;	// LineDB
      L     1;	// code.Warning
      JC    I103;
//-Loaded-------------------------------
I1N5: L     #TmpWord;	// bit_main_status
      L     2#100000000001;	// mask with loaded code
      AW;
      JZ    I1N6;
      A     #PCRead.Status.StaLoaded;	// LineDB
      L     5;	// code.Loaded
      JC    I103;
//-NoSubState---------------------------
I1N6: L     0;	// code.NoSubState
// 
//=Build InfoCode=======================
I103: L     #TmpInt;	// MainInfoCode
      +I;	// Add SubInfoCode
      T     #PCRead.InfoCode;	//-->LineDB
      BEU;
I100: NOP   0;
NETWORK
TITLE = Sub1061: GC GGRs status colour WinCoS
//Inputs :
// LineDB.VarTemp.InOutValue3 = Relevant Groups
//
//Outputs:
// no
//
      L     #InCode;
      L     1061;
      <>I;
      JC    GC00;
//-Init--- 
      L     #VarTemp.InOutValue3;	//[2.3]
      T     #TmpDInt;	//[2.3]
      L     #VarTemp.InOutValue4;	//[3.0]
      T     #tmpDInt2;	//[3.0]
      L     0;
      LAR1  P##tmpLin_GenGrpCoulorCode;
      T     LW [AR1,P#0.0];	//Reset tmpLin_GenGrpCoulorCode
      OPN   DB 9;
//============================================
//Loop Section 
//============================================
      L     DB9.DBW 0;	//ParByteNoSecDB
      SLD   3;
GCLS: T     #DB9SecArray;
      OPN   DB 9;
//-----------------------------------
//Test End Of Array DB9.Sectio
      L     W#16#FFFF;
      L     DBW [#DB9SecArray];	// DB9.Section[x].DBNr
      ==I;
      JC    GCOT;	//-> Return
//-----------------------------------
//Read pointer to section interface
      T     #tmpSecDB;
      L     0;
      ==I;
      JC    GCNS;	//--> IF DBNr= 0 THEN  Next section
//-----------------------------------
//Start address Interface GroupControl in section
      LAR1  #DB9SecArray;
      OPN   DB 9;
      L     DBW [AR1,P#2.0];	//  DB9.Section[x].DBB
      SLD   3;
      T     #tmpAddrGrInterfaceSec;	//-->Pointer to instance in section DB
//-----------------------------------
//Check if section DB belongs to actual process line
      OPN   DI [#tmpSecDB];	// Call Section DB
      L     #Para.ParLineDB_ParFirstSecDB;	// S_DB
      L     #tmpLineDB;
      <>I;
      JC    GCNS;	//-->Next section
//-----------------------------------
//Start address Interface GroupControl in section
//========================================================= 
//Section[x]
//---------- 
//-Evaluate involved groups--- 
      LAR1  #tmpAddrGrInterfaceSec;	// Pointer to instance in section DB
      L     DID [AR1,P#52.0];	// SEC.Gr.OutSelected [08..01/16..09//24..17/32..25]
      L     #TmpDInt;	// USW selected relevant GGR [2.3]
      AD;
      T     #tmpRelevantGroups32_1;	//--> Mask of relevant GGR
      L     DID [AR1,P#56.0];	// SEC.Gr.OutSelected [40..33/48..41//56..49/64..57] [3.0]
      L     #tmpDInt2;	// USW selected relevant GGR [2.3]                   [3.1]
      AD;	//                                                   [3.0]
      T     #tmpRelevantGroups64_33;	//--> Mask of relevant GGR                           [3.0]
//-No State----------------------------------
      L     #tmpRelevantGroups32_1;	// Mask of relevant GGR
      L     2#0;	// No group selected
      ==D;
      A(;	//                       [3.0]
      L     #tmpRelevantGroups64_33;	// Mask of relevant GGR  [3.0]
      L     2#0;	// No group selected     [3.0]
      ==D;	//                       [3.0]
      );	//                       [3.0]
      L     2#1;	// GenGrpStateCode.lightGrey (DB321.DBX x.0)
      JC    GC01;
//-Fault-------------------------------
      L     #tmpRelevantGroups32_1;	// Mask of relevant GGR
      L     DB9.DBD 530;	// InFault [08..01/16..09//24..17/32..25]
      AD;
      L     0;
      <>D;
      O(;	//                                        [3.0]
      L     #tmpRelevantGroups64_33;	// Mask of relevant GGR                   [3.0]
      L     DB9.DBD 534;	// InFault [40..33/48..41//56..49/64..57] [3.0]
      AD;	//                                        [3.0]
      L     0;	//                                        [3.0]
      <>D;	//                                        [3.0]
      );	//                                        [3.0]
      L     2#10000;	// GenGrpStateCode.red (DB321.DBX x.4)
      JC    GC01;
//-Warning--------------------------------
      L     #tmpRelevantGroups32_1;	// Mask of relevant GGR
      L     DB9.DBD 570;	// InWarning [08..01/16..09//24..17/32..25]
      AD;
      L     0;
      <>D;
      O(;	//                                          [3.0]
      L     #tmpRelevantGroups64_33;	// Mask of relevant GGR                     [3.0]
      L     DB9.DBD 574;	// InWarning [40..33/48..41//56..49/64..57] [3.0]
      AD;	//                                          [3.0]
      L     0;	//                                          [3.0]
      <>D;	//                                          [3.0]
      );	//                                          [3.0]
      L     2#1000;	// GenGrpStateCode.magenta (DB321.DBX x.3)
      JC    GC01;
//-Else------------------------------
      L     2#100;	// GenGrpStateCode.darkGreen (DB321.DBX x.2)
GC01: LAR1  P##tmpSec_GenGrpCoulorCode;
      T     LB [AR1,P#0.0];	//-->tmpGenGrpCoulorCode  
//=================================================================
// Add Section-State to Line-State
//====================================================================
      OPN   DI [#tmpLineDB];	// Call L-DB
//-Fault--------------------------------
      A     #tmpLin_GenGrpCoulorCode.red;
      O     #tmpSec_GenGrpCoulorCode.red;
      L     2#10000;	// GenGrpCoulorCode.Fault 
      JC    GC02;
//-Warning------------------------------
      A     #tmpLin_GenGrpCoulorCode.magenta;
      O     #tmpSec_GenGrpCoulorCode.magenta;
      L     2#1000;	// GenGrpCoulorCode.Warning
      JC    GC02;
//-Started------------------------------
      A     #tmpLin_GenGrpCoulorCode.darkGreen;
      O     #tmpSec_GenGrpCoulorCode.darkGreen;
      L     2#100;	// GenGrpCoulorCode.Started
      JC    GC02;
//-No State-----------------------------
      L     2#1;	// GenGrpCoulorCode.lightGrey 
//-Save state---
GC02: LAR1  P##tmpLin_GenGrpCoulorCode;
      T     LB [AR1,P#0.0];	//Reset tmpLin_GenGrpCoulorCode [2.4]
//=== Call Next Section  =====================================
GCNS: L     #DB9SecArray;
      L     P#4.0;
      +D;	// Pointer to next section
      JU    GCLS;
GCOT: OPN   DI [#tmpLineDB];
      LAR1  P##tmpLin_GenGrpCoulorCode;
      L     LB [AR1,P#0.0];	//Reset tmpLin_GenGrpCoulorCode [2.4]
      T     #PCRead.SectionState;	//->LineDB  PCRead.GenGrpColorCode
// 
      BEU;
// 
GC00: NOP   0;
NETWORK
TITLE = Sub1062: MC Maintenance status colour WinCoS
//Inputs :
// LineDB.VarTemp.InOutValue3 = Relevant Groups
//
//Outputs:
// Colour code on line-DB
//
      L     #InCode;
      L     1062;
      <>I;
      JC    MC00;
//-Init--- 
      L     #VarTemp.InOutValue3;	//[2.3]
      T     #TmpDInt;	//[2.3]
      L     0;
      LAR1  P##tmpLin_GenGrpCoulorCode;
      T     LW [AR1,P#0.0];	//Reset tmpLin_GenGrpCoulorCode
      OPN   DB 9;
//============================================
//Loop Section 
//============================================
      L     DB9.DBW 0;	//ParByteNoSecDB
      SLD   3;
MCLS: T     #DB9SecArray;
      OPN   DB 9;
//-----------------------------------
//Test End Of Array DB9.Sectio
      L     W#16#FFFF;
      L     DBW [#DB9SecArray];	// DB9.Section[x].DBNr
      ==I;
      JC    MCOT;	//-> Return
//-----------------------------------
//Read pointer to section interface
      T     #tmpSecDB;
      L     0;
      ==I;
      JC    MCNS;	//--> IF DBNr= 0 THEN  Next section
//-----------------------------------
//Start address Interface GroupControl in section
      LAR1  #DB9SecArray;
      OPN   DB 9;
      L     DBW [AR1,P#2.0];	//  DB9.Section[x].DBB
      SLD   3;
      T     #tmpAddrGrInterfaceSec;	//-->Pointer to instance in section DB
//-----------------------------------
//Check if section DB belongs to actual process line
      OPN   DI [#tmpSecDB];	// Call Section DB
      L     #Para.ParLineDB_ParFirstSecDB;	// S_DB
      L     #tmpLineDB;
      <>I;
      JC    MCNS;	//-->Next section
//-----------------------------------
//Start address Interface GroupControl in section
//========================================================= 
//Section[x]
//---------- 
//-Evaluate involved groups--- 
      LAR1  #tmpAddrGrInterfaceSec;	// Pointer to instance in section DB
      L     DID [AR1,P#52.0];	// SEC.Gr.OutSelected [08..01/16..09//24..17/32..25]
      L     #TmpDInt;	// USW selected relevant GGR [2.3]
      AD;
      T     #tmpRelevantGroups32_1;	//--> Mask of relevant GGR
//-No State----------------------------------
      L     #tmpRelevantGroups32_1;	// Mask of relevant GGR
      L     2#0;	// No group selected
      ==D;
      L     2#1;	// GenGrpStateCode.lightGrey (DB321.DBX x.0)
      JC    MC01;
//-Fault-------------------------------
      L     #tmpRelevantGroups32_1;	// Mask of relevant GGR
      L     DB9.DBD 530;	// InFault [08..01/16..09//24..17/32..25]
      AD;
      L     0;
      <>D;
      L     2#10000;	// GenGrpStateCode.red (DB321.DBX x.4)
      JC    MC01;
//-Warning--------------------------------
      L     #tmpRelevantGroups32_1;	// Mask of relevant GGR
      L     DB9.DBD 570;	// InWarning [08..01/16..09//24..17/32..25]
      AD;
      L     0;
      <>D;
      L     2#1000;	// GenGrpStateCode.magenta (DB321.DBX x.3)
      JC    MC01;
//-Else------------------------------
      L     2#100;	// GenGrpStateCode.darkGreen (DB321.DBX x.2)
MC01: LAR1  P##tmpSec_GenGrpCoulorCode;
      T     LB [AR1,P#0.0];	//-->tmpGenGrpCoulorCode  
//=================================================================
// Add Section-State to Line-State
//====================================================================
      OPN   DI [#tmpLineDB];	// Call L-DB
//-Fault--------------------------------
      A     #tmpLin_GenGrpCoulorCode.red;
      O     #tmpSec_GenGrpCoulorCode.red;
      L     2#10000;	// GenGrpCoulorCode.Fault 
      JC    MC02;
//-Warning------------------------------
      A     #tmpLin_GenGrpCoulorCode.magenta;
      O     #tmpSec_GenGrpCoulorCode.magenta;
      L     2#1000;	// GenGrpCoulorCode.Warning
      JC    MC02;
//-Started------------------------------
      A     #tmpLin_GenGrpCoulorCode.darkGreen;
      O     #tmpSec_GenGrpCoulorCode.darkGreen;
      L     2#100;	// GenGrpCoulorCode.Started
      JC    MC02;
//-No State-----------------------------
      L     2#1;	// GenGrpCoulorCode.lightGrey 
//-Save state---
MC02: LAR1  P##tmpLin_GenGrpCoulorCode;
      T     LB [AR1,P#0.0];	//Reset tmpLin_GenGrpCoulorCode [2.4]
//=== Call Next Section  =====================================
MCNS: L     #DB9SecArray;
      L     P#4.0;
      +D;	// Pointer to next section
      JU    MCLS;
MCOT: OPN   DI [#tmpLineDB];
      LAR1  P##tmpLin_GenGrpCoulorCode;
      L     LB [AR1,P#0.0];	//Reset tmpLin_GenGrpCoulorCode [2.4]
      T     #PCRead.Value7;	//->LineDB  PCRead.MaintenanceGrpColorCode
// 
      BEU;
// 
MC00: NOP   0;
NETWORK
TITLE = Sub2001: SC Section commands
//Open DB = Section DB
//
//Inputs:
// SectionDB.VarTemp.InOutValue3 = Precutoff weight
      L     #InCode;
      L     2001;
      <>I;
      JC    SC00;
//--- FKT.immediate_stop---------------
      A     #PCRead.Status.StaHWStop;
      S     #ToSSW.Func.CmdImmediateStop;
//--- FKT.empty_section ---------------
      A     #JobAc.StaBatch.StaEmptyingBatch;
      S     #ToSSW.Func.CmdFeedOff;
      A     #JobAc.StaBatch.StaEmptyingBatch;
      A     #PCRead.Step.StActive;
      S     #ToSSW.Func.CmdSequenzStop;
      S     #PCRead.Status.StaLoaded;
//--- FKT.step_mode -------------------
      A     #PCRead.Status.StaStep;
      S     #ToSSW.Func.CmdFeedOff;
      A     #ToSSW.InfStarted;
//[4.2]      U     #PCRead.Step.StActive
      AN    #PCRead.Step.StPassive;	//[4.2]
      AN    #PCRead.Step.StIdling;	//[4.2]
      AN    #PCRead.Step.StWait;	//[4.2]
      S     #ToSSW.Func.CmdStepOff;
//--- FKT.sequnce_stop ----------------
      A(;
      L     #JobNom.FeedingTime;
      L     #JobAc.FeedingTime;
      <=I;
      A(;
      L     0;
      L     #JobNom.FeedingTime;
      <>I;
      );
      );
      O(;
      L     #JobNom.JobWeight;
      L     #VarTemp.InOutValue3;	// Prestop weight  [1.7]
      -D;	//                 [1.7]
      L     #JobAc.JobWeight;
      <=D;
      A(;
      L     0;
      L     #JobNom.JobWeight;
      <>D;
      );
      );
      A     #PCRead.Step.StActive;
      S     #ToSSW.Func.CmdSequenzStop;
      BEU;
SC00: NOP   0;
NETWORK
TITLE = Sub2002: SS Extended section commands
//Called by line controler subroutines, with opened L-DB
      L     #InCode;
      L     2002;
      <>I;
      JC    SS01;
      L     #PCWrite.Value1;	// PCWrite.ExtFuncOn 
      T     #PCRead.ExtFuncOn;
//-Update ExtStatus------------------------
      L     #PCRead.ExtStatus;	// ExtStatus
      L     #PCWrite.Value1;	// PCWrite.ExtFuncOn 
      OD;	// 
      L     #PCWrite.Value2;	// PCWrite.ExtFuncOff 
      INVD;	//  
      AD;	//  
      T     #PCRead.ExtStatus;	//->ExtStatus
//Reset on commands 
      L     0;
      T     #PCWrite.Value1;	// PCWrite.ExtFuncOn 
//Reset off commands 
      L     0;
      T     #PCWrite.Value2;	// PCWrite.ExtFuncOff 
      BEU;
SS01: NOP   0;
NETWORK
TITLE = Sub2003:SI Section init
//Called by section controler subroutines
//
//Open DB = Section DB
//
//Inputs :
// no
//Outputs:
// no
//
      L     #InCode;
      L     2003;
      <>I;
      JC    SI00;
//-FKT.immediate_stop------------------
//[3.4]      SET   
//[3.4]      R     #PCRead.Status.StaImmediateStop
//-FKT.feeding_time--------------------
      L     0;
      T     #JobAc.FeedingTime;
      BEU;
SI00: NOP   0;
NETWORK
TITLE = Sub2004: FT Feeding time
//Called by section controler subroutines
//Open DB = Section DB
//
//Inputs :
// no
//Outputs:
// no
//
      L     #InCode;
      L     2004;
      <>I;
      JC    FT00;
      A     #PCRead.State.StFeeding;
      A     "SYS_Scan0_Tick1min";	//"SYS_Scan0_Tick1min"
      JCN   FT02;
      L     32767;
      L     #JobAc.FeedingTime;
      <=I;
      JC    FT01;	//If Time = maxValue then set to 0
      +     1;
      T     #JobAc.FeedingTime;
      BEU;
FT01: L     1;
      T     #JobAc.FeedingTime;
FT02: BEU;
FT00: NOP   0;
NETWORK
TITLE = Sub2051: ST Section status text and colour
//Called by section controler subroutines
//Open DB = Section DB
//
//Inputs :
// no
//Outputs:
// no
//
      L     #InCode;
      L     2051;
      <>I;
      JC    ST00;
//=Build auxiliary status===============
//-Passive------------------------------
      A     #PCRead.Step.StPassive;
      L     2#1;
      L     100;	// code.st_passiv
      JC    ST01;
//-Ready--------------------------------
      A     "SYS_infLog0";	// !! not used !!
      L     2#10;
      L     200;	// code.st_ready
      JC    ST01;
//-Available test-----------------------
      A     #PCRead.Step.StWait;
      L     2#100;
      L     300;	// code.st_available_test
      JC    ST01;
//-Start Warning------------------------
      A     #PCRead.Status.StaStartwarning;
      L     2#1000;
      L     400;	// code.st_startwarning
      JC    ST01;
//-Starting-----------------------------
      A     #PCRead.Step.StActive;
      A     #PCRead.State.StStarting;
      L     2#10000;
      L     500;	// code.st_starting
      JC    ST01;
//-Suspended----------------------------
      A     #PCRead.Step.StActive;
      A     #PCRead.State.StStarted;
      AN    #PCRead.State.StFeeding;
      L     2#100000;
      L     600;	// code.st_suspended
      JC    ST01;
//-Running------------------------------
      A     #PCRead.Step.StActive;
      A     #PCRead.State.StFeeding;
      L     2#1000000;
      L     700;	// code.st_running
      JC    ST01;
//-Wait---------------------------------
      A     #PCRead.Step.StReady;
      AN    #PCRead.Step.StEmptying;
      L     2#10000000;
      L     800;	// code.st_wait
      JC    ST01;
//-Emptying-----------------------------
      A     #PCRead.Step.StEmptying;
      AN    #ToSSW.InfReleaseEmptyingTime;
      AN    #PCRead.State.StStopped;
      L     2#100000000;
      L     900;	// code.st_emtying
      JC    ST01;
//-Emptying active----------------------
      A     #PCRead.Step.StEmptying;
      A     #ToSSW.InfReleaseEmptyingTime;
      AN    #PCRead.State.StStopped;
      L     2#1000000000;
      L     1000;	// code.st_emptying_activ
      JC    ST01;
//-Registration-------------------------
      A     #PCRead.Step.StEmptied;
      L     2#10000000000;
      L     1100;	// code.st_registration
      JC    ST01;
//-Idling-------------------------------
      A     #PCRead.Step.StIdling;
      L     2#100000000000;
      L     1200;	// code.st_idling
      JC    ST01;
//-Stopping-----------------------------
      A     #PCRead.State.StStopping;
      L     2#1000000000000;
      L     1300;	// code.st_stopping
      JC    ST01;
//-Stopped------------------------------
      AN    #PCRead.Step.StPassive;
      A     #PCRead.State.StStopped;
      L     2#10000000000000;
      L     1400;	// code.st_stopped
      JC    ST01;
//-No State-----------------------------
      L     2#0;
      L     0;	// code.st_no_state
ST01: T     #TmpInt;
      TAK;
      T     #TmpWord;
//==Status text=========================
//-Fault--------------------------------
      L     #TmpWord;
      L     2#11011111111100;	// status with fault code
      AW;
      JZ    ST11;
      A     #PCRead.Fault.EsMech;
      L     2;	// code.st_fault
      JC    ST02;
//-Warning------------------------------
ST11: L     #TmpWord;
      L     2#11011111111000;	// status with warning code
      AW;
      JZ    ST12;
      A     #PCRead.Fault.EsWarning;
      L     1;	// code.st_warning
      JC    ST02;
//-Restart------------------------------
ST12: L     #TmpWord;
      L     2#11000011110000;	// status with restart code
      AW;
      JZ    ST13;
      AN    #PCRead.Status.StaAutostart;
      L     3;	// code.st_restart
      JC    ST02;
//-Step mode----------------------------
ST13: L     #TmpWord;
      L     2#11000000111111;	// status with step_mode code
      AW;
      JZ    ST14;
      A     #PCRead.Status.StaStep;
      L     4;	// code.st_step_mode
      JC    ST02;
//-Loaded-------------------------------
ST14: L     #TmpWord;
      L     2#11000000000001;	// status with loaded code
      AW;
      JZ    ST15;
      A     #PCRead.Status.StaLoaded;
      L     5;	// code.st_loaded
      JC    ST02;
//-Mixing-------------------------------
ST15: L     #TmpWord;
      L     2#100000;	// status with mixing code
      AW;
      JZ    ST03;
      A     "SYS_infLog0";	// !!! not used !!!
      L     6;	// code.st_mixing
      JC    ST02;
      JU    ST03;
//-Build real text status---------------
ST02: L     #TmpInt;
      +I;
      T     #TmpInt;
//==Status colour=======================
//-Fault--------------------------------
ST03: L     #TmpWord;
      L     2#11011111111100;	// mask text code
      AW;
      JZ    ST31;
      A     #PCRead.Fault.EsMech;
      O     #PCRead.Fault.EsDosing;
      L     2#1000000000000000;	// additional_code.red
      JC    ST04;
//-Warning------------------------------
ST31: L     #TmpWord;
      L     2#11011111111000;	// mask text code
      AW;
      JZ    ST32;
      A     #PCRead.Fault.EsWarning;
      L     2#100000000000000;	// additional_code.magenta
      JC    ST04;
//-Ready for restart--------------------
ST32: L     #TmpWord;
      L     2#11011111111000;	// mask text code
      AW;
      JZ    ST33;
      A(;
      O     #PCRead.Step.StActive;
      O     #PCRead.Step.StReady;
      O     #PCRead.Step.StEmptying;
      O     #PCRead.Step.StEmptied;
      );
      AN    #PCRead.Status.StaAutostart;
      O;
      A     #PCRead.Status.StaFeedOff;
      A     #PCRead.Step.StActive;
      A     #PCRead.State.StStarted;
      AN    #PCRead.State.StFeeding;
      L     2#10000000;	// additional_code.tuerkis
      JC    ST04;
//-Step mode----------------------------
ST33: L     #TmpWord;
      L     2#11000000111111;	// mask text code
      AW;
      JZ    ST34;
      AN    #PCRead.Step.StPassive;
      A     #PCRead.Status.StaStep;
      L     2#100000;	// additional_code.brown
      JC    ST04;
//-Occupied-----------------------------
ST34: L     #TmpWord;
      L     2#100000000001;	// mask text code
      AW;
      JZ    ST35;
      A     #PCRead.Status.StaLoaded;
      L     2#1000000;	// additional_code.orange
      JC    ST04;
//-Starting-----------------------------
ST35: L     #TmpWord;
      L     2#11100;	// mask text code
      AW;
      JZ    ST36;
      L     2#10000000000000;	// code.light green
      JU    ST04;
//-Suspended----------------------------
ST36: L     #TmpWord;
      L     2#10100000;	// mask text code
      AW;
      JZ    ST37;
      L     2#1000000000000;	// code.green
      JU    ST04;
//-Running------------------------------
ST37: L     #TmpWord;
      L     2#1000000;	// mask text code
      AW;
      JZ    ST38;
      L     2#100000000000;	// code.dark green
      JU    ST04;
//-Emptying/Emptied---------------------
ST38: L     #TmpWord;
      L     2#11100000010;	// mask text code
      AW;
      JZ    ST39;
      L     2#10000000000;	// code.blue
      JU    ST04;
//-Stopping/Stopped---------------------
ST39: L     #TmpWord;
      L     2#11000000000000;	// mask text code
      AW;
      JZ    ST40;
      L     2#1000000000;	// code.yellow
      JU    ST04;
//-Passive/Idling-----------------------
ST40: L     #TmpWord;
      L     2#100000000001;	// mask text code
      AW;
      JZ    ST41;
      L     2#100000000;	// code.white
      JU    ST04;
//-Default------------------------------
ST41: L     2#100000000;	// code.weiss (default)
//=Data to MELE=========================
ST04: T     #TmpWord;	// --> Section colour state
//Check if any value changed PCRead.LineInfoCode
      L     #PCRead.InfoCode;
      ==I;
      A(;
      L     #TmpInt;
      L     #PCRead.SectionState;
      ==I;
      );
      BEC;
      S     #ChangeBit.CBit1;
      L     #TmpWord;	// Save section color status    
      T     #PCRead.InfoCode;
      L     #TmpInt;	// Save section text status
      T     #PCRead.SectionState;
      BEU;
ST00: NOP   0;
NETWORK
TITLE = Sub2055: SI Section info code : WinCoS
//Called by section controler subroutines
//
//Open DB = Section DB
//Inputs :
// no
//Outputs:
// no
//
      L     #InCode;
      L     2055;
      <>I;
      JC    I200;
// 
//=Build MainInfoCode===================
//-Fault--------------------------------
      A     #PCRead.Fault.EsMech;
      O     #PCRead.Fault.EsDosing;
      O     #PCRead.Fault.EsBatchSize;
      O     #PCRead.Fault.EsRefillLevel;
      AN    #PCRead.Step.StPassive;
      AN    #PCRead.Step.StIdling;
      L     2#100000000000000;
      L     1500;	// code.st_fault
      JC    I201;
//-Passive------------------------------
      A     #PCRead.Step.StPassive;
      L     2#1;
      L     100;	// code.st_passiv
      JC    I201;
//-Ready--------------------------------
      CLR;	// !! not used !!
      L     2#10;
      L     200;	// code.st_ready
      JC    I201;
//-Available test-----------------------
      A     #PCRead.Step.StWait;
      L     2#100;
      L     300;	// code.st_available_test
      JC    I201;
//-Start Warning------------------------
      A     #PCRead.Status.StaStartwarning;	// S.PCRead.Status.StaStartwarning
      L     2#1000;
      L     400;	// code.st_startwarning
      JC    I201;
//-Starting-----------------------------
      A     #PCRead.Step.StActive;
      AN    #ToSSW.InfStarted;
      AN    #PCRead.State.StStopped;
      AN    #PCRead.State.StStopping;
//    U     PCRead.State.StStarting    
      L     2#10000;
      L     500;	// code.st_starting
      JC    I201;
//-Suspended----------------------------
      A     #PCRead.Step.StActive;
      A     #PCRead.State.StStarted;
      AN    #PCRead.State.StFeeding;
      L     2#100000;
      L     600;	// code.st_suspended
      JC    I201;
//-Running------------------------------
      A     #PCRead.Step.StActive;
      A     #PCRead.State.StFeeding;
      L     2#1000000;
      L     700;	// code.st_running
      JC    I201;
//-Wait---------------------------------
      A     #PCRead.Step.StReady;
      AN    #PCRead.Step.StEmptying;
      L     2#10000000;
      L     800;	// code.st_wait
      JC    I201;
//-Emptying-----------------------------
      A     #PCRead.Step.StEmptying;
      AN    #ToSSW.InfReleaseEmptyingTime;
      AN    #PCRead.State.StStopped;
      L     2#100000000;
      L     900;	// code.st_emtying
      JC    I201;
//-Emptying active----------------------
      A     #PCRead.Step.StEmptying;
      A     #ToSSW.InfReleaseEmptyingTime;
      AN    #PCRead.State.StStopped;
      L     2#1000000000;
      L     1000;	// code.st_emptying_activ
      JC    I201;
//-Registration-------------------------
      A     #PCRead.Step.StEmptied;
      L     2#10000000000;
      L     1100;	// code.st_registration
      JC    I201;
//-Idling-------------------------------
      A     #PCRead.Step.StIdling;
      L     2#100000000000;
      L     1200;	// code.st_idling
      JC    I201;
//-Stopping-----------------------------
      A     #PCRead.State.StStopping;
      L     2#1000000000000;
      L     1300;	// code.st_stopping
      JC    I201;
//-Stopped------------------------------
      AN    #PCRead.Step.StPassive;
      A     #PCRead.State.StStopped;
      L     2#10000000000000;
      L     1400;	// code.st_stopped
      JC    I201;
//-No State-----------------------------
      L     2#0;
      L     0;	// code.st_no_state
I201: T     #TmpInt;
      TAK;
      T     #TmpWord;
//=Build SubInfoCode====================
//-DPFault------------------------------
      L     #TmpWord;	// bit_main_status
      L     2#111111111111111;	// mask with restart code
      AW;
      JZ    I2I1;
      A     #PCRead.Status.StaDPFault;
      L     7;	// code.dpfault
      JC    I202;
//-Restart------------------------------
I2I1: L     #TmpWord;
      L     2#111011111111000;	// status with restart code
      AW;
      JZ    I212;
      A     #PCRead.Status.StaImmediateStop;
      O     #PCRead.Status.StaTransferOff;
      O     #PCRead.Status.StaFeedOff;
      AN    #PCRead.Status.StaStep;
      ON    #PCRead.Status.StaAutostart;
      L     3;	// code.st_restart
      JC    I202;
//-Step mode----------------------------
I212: L     #TmpWord;
      L     2#111000000111111;	// status with step_mode code
      AW;
      JZ    I213;
      A     #PCRead.Status.StaStep;
      L     4;	// code.st_step_mode
      JC    I202;
//-Hold---------------------------------
I213: L     #TmpWord;
      L     2#111100001111111;	// status with step_mode code
      AW;
      JZ    I214;
      A     #PCRead.Status.StaHold;
      L     6;	// code.st_step_mode
      JC    I202;
//-Warning------------------------------
I214: L     #TmpWord;
      L     2#111011111111000;	// status with warning code
      AW;
      JZ    I215;
      A     #PCRead.Fault.EsWarning;
      L     1;	// code.st_warning
      JC    I202;
//-Loaded-------------------------------
I215: L     #TmpWord;
      L     2#100000000001;	// status with loaded code
      AW;
      JZ    I216;
      A     #PCRead.Status.StaLoaded;	// S.PCRead.Status.StaLoaded
      L     5;	// code.st_loaded
      JC    I202;
//-NoSubState---------------------------
I216: L     0;	// code.NoSubState
// 
//=Build InfoCode=======================
I202: L     #TmpInt;	// MainInfoCode
      +I;	// Add SubInfoCode
      T     #PCRead.InfoCode;
      BEU;
I200: NOP   0;
NETWORK
TITLE = Sub2071: PIC FU: Section info code
//Called by section controler subroutines
//
//Open DB = Section DB
//Inputs :
// no
//Outputs:
// no
//
      L     #InCode;
      L     2071;
      <>I;
      JC    I300;
// Reset 
      L     0;
      LAR1  P##tmpUserState;
      T     LW [AR1,P#0.0];
//-StFault
      A(;
      O     #PCRead.Fault.EsEmpty;
      O     #PCRead.Fault.EsFull;
      AN    #PCRead.Step.StPassive;
      AN    #PCRead.Step.StEmptying;
      AN    #PCRead.Step.StEmptied;
      AN    #PCRead.Step.StIdling;
      );
      O     #PCRead.Fault.EsWayConflict;
      O     #PCRead.Fault.EsMech;
      O     #PCRead.Fault.EsDosing;
      O     #PCRead.Fault.EsInterrupt;
      O     #PCRead.Fault.EsBatchSize;
      =     #tmpUserState.stEmptying;
      JC    Tran;
//-StPassive
      A     #PCRead.Step.StPassive;
      A     #PCRead.State.StStopped;
      AN    #PCRead.Status.StaHold;
      AN    #PCRead.Status.StaHand;
      AN    #PCRead.Status.StaStep;
      =     #tmpUserState.stEmptied;
      JC    Tran;
//-StWait
      A     #PCRead.Step.StWait;
      AN    #PCRead.Status.StaHold;
      AN    #PCRead.Status.StaHand;
      AN    #PCRead.Status.StaStep;
      =     #tmpUserState.stIdling;
      JC    Tran;
//-StStarting--
      A     #PCRead.Step.StActive;
      A     #PCRead.State.StStarting;
      AN    #PCRead.Status.StaHold;
      AN    #PCRead.Status.StaHand;
      AN    #PCRead.Status.StaStep;
      =     #tmpUserState.stFault;
      JC    Tran;
//-StStarted--
      A     #PCRead.Step.StActive;
      A     #PCRead.State.StStarted;
      AN    #PCRead.Status.StaHold;
      AN    #PCRead.Status.StaHand;
      AN    #PCRead.Status.StaStep;
      =     #tmpUserState.stHand;
      JC    Tran;
//-StStopping--
      A     #PCRead.Step.StActive;
      A     #PCRead.State.StStopping;
      AN    #PCRead.Status.StaHold;
      AN    #PCRead.Status.StaHand;
      AN    #PCRead.Status.StaStep;
      =     #tmpUserState.stHold;
      JC    Tran;
//-StStopped--
      A     #PCRead.Step.StActive;
      A     #PCRead.State.StStopped;
      AN    #PCRead.Status.StaHold;
      AN    #PCRead.Status.StaHand;
      AN    #PCRead.Status.StaStep;
      =     #tmpUserState.stStep;
      JC    Tran;
//-StFeeding--
      A     #PCRead.Step.StActive;
      A     #PCRead.State.StFeeding;
      AN    #PCRead.Status.StaHold;
      AN    #PCRead.Status.StaHand;
      AN    #PCRead.Status.StaStep;
      AN    #PCRead.Status.StaEndOfJob;
      =     #tmpUserState.stPassive;
      JC    Tran;
//-StReady--
      A     #PCRead.Step.StReady;
      AN    #PCRead.Status.StaHold;
      AN    #PCRead.Status.StaHand;
      AN    #PCRead.Status.StaStep;
      =     #tmpUserState.stWait;
      JC    Tran;
//-StEmptying--
      A     #PCRead.State.StFeeding;
      A     #PCRead.Status.StaEndOfJob;
      O     #PCRead.Step.StEmptying;
      AN    #PCRead.Status.StaHold;
      AN    #PCRead.Status.StaHand;
      AN    #PCRead.Status.StaStep;
      =     #tmpUserState.stStarting;
      JC    Tran;
//-StEmptied--
      A     #PCRead.Step.StEmptied;
      AN    #PCRead.Status.StaHold;
      AN    #PCRead.Status.StaHand;
      AN    #PCRead.Status.StaStep;
      =     #tmpUserState.stStarted;
      JC    Tran;
//-StIdling--
      A     #PCRead.Step.StIdling;
      AN    #PCRead.Status.StaHold;
      AN    #PCRead.Status.StaHand;
      AN    #PCRead.Status.StaStep;
      =     #tmpUserState.stStopping;
//-StHand--
      A     #PCRead.Status.StaHand;
      AN    #PCRead.Status.StaHold;
      AN    #PCRead.Status.StaStep;
      =     #tmpUserState.stStopped;
      JC    Tran;
//-StHold--
      A     #PCRead.Status.StaHold;
      AN    #PCRead.Status.StaHand;
      AN    #PCRead.Status.StaStep;
      =     #tmpUserState.stFeeding;
      JC    Tran;
//-StStep--
      A     #PCRead.Status.StaStep;
      AN    #PCRead.Status.StaHold;
      AN    #PCRead.Status.StaHand;
      =     #tmpUserState.stReady;
      JC    Tran;
//Store New Code
Tran: L     #PCRead.SectionState;
      LAR1  P##tmpUserState;
      L     LW [AR1,P#0.0];
      T     #PCRead.SectionState;
// Changebit
      <>I;
      S     #ChangeBit.CBit1;
      BEU;
I300: NOP   0;
NETWORK
TITLE = End of block
      BE;
END_FUNCTION_BLOCK

FUNCTION_BLOCK "TON_BREAK"	// FB 1704
TITLE = TON with break possibility
//COPYRIGHT:    (C) 2004 BY  BUHLER LTD.
//                           CH-9240 UZWIL  SWITZERLAND
//
//PRODUCT:      STD_MU664    
//
//TITLE:        IEC-TON timer with break functionality
//              
//              IEC-TON Zeitverzögerung mit Unterbrechungsfunktionalität
//
//    
//
//--------------------------------------------------------------------------------
//
//IDENT:        AUTOR:              DEPT:                              DATE:
//STD_FB1704.1.0Ph. Engler          MU664                              24-May-2004
//              1st Release
//
//--------------------------------------------------------------------------------
//
//PURPOSE:      
//
//RESTRICTIONS:
//
//--------------------------------------------------------------------------------
//
AUTHOR : PE
FAMILY : STD
VERSION : 1.0
VAR_INPUT
  IN : BOOL ;	//Start timer
  BREAK : BOOL ;	//Interrupt timer
  PT : INT ;	//Time delay in seconds
END_VAR
VAR_OUTPUT
  Q : BOOL ;	//Time elapsed
  ET : INT ;	//Elapsed time in seconds
  RT : INT ;	//Rest time in seconds
END_VAR
VAR
  EdgeIN : BOOL ;
  CNT : SFB 2;
END_VAR
BEGIN
NETWORK
TITLE = Inputs
      L     #PT;
      T     #CNT.PV;
// 
      AN    #IN;
      =     #CNT.R;
// 
      A     #IN;
      AN    #BREAK;
      A     "SYS_Scan0_Tick1s";
      AN    #CNT.QU;
      =     #CNT.CU;
NETWORK
TITLE = Call counter
      CALL  #CNT;
NETWORK
TITLE = Outputs
      L     #CNT.CV;
      T     #ET;
      L     #CNT.PV;
      TAK;
      -I;
      T     #RT;
// 
      A     #CNT.QU;
      =     #Q;
NETWORK
TITLE = End of block
      BE;
END_FUNCTION_BLOCK

FUNCTION_BLOCK "T_BREAK"	// FB 1706
TITLE = TON with break possibility
//COPYRIGHT:    (C) 2004 BY  BUHLER LTD.
//                           CH-9240 UZWIL  SWITZERLAND
//
//PRODUCT:      STD_MU664    
//
//TITLE:        IEC-TON timer with break functionality
//              
//              IEC-TON Zeitverzögerung mit Unterbrechungsfunktionalität
//
//    
//
//--------------------------------------------------------------------------------
//
//IDENT:         AUTOR:              DEPT:                             DATE:
//STD_FB1706.2.0 Ph. Engler          MU664                             24-May-2004
//               Support for TON and TOF type
//STD_FB1706.1.0 Ph. Engler          MU664                             24-May-2004
//               1st Release
//
//--------------------------------------------------------------------------------
//
//PURPOSE:      
//
//RESTRICTIONS:
//
//--------------------------------------------------------------------------------
//
AUTHOR : PE
FAMILY : STD
VERSION : 2.0
VAR_INPUT
  IN : BOOL ;	//Start timer
  BREAK : BOOL ;	//Interrupt timer
  TON : BOOL ;	//Type of timer TON->0 = TOF
  ParRestart : BOOL ;
  ParRecalc : BOOL ;
  PT : INT ;	//Time delay in seconds
END_VAR
VAR_OUTPUT
  Q : BOOL ;	//Time elapsed
  ET : DINT ;	//Elapsed time in seconds
  RT : INT ;	//Rest time in seconds
END_VAR
VAR
  EdgeIN : BOOL ;
  CNT : SFB 2;
  Par : STRUCT
   Spare01 : BOOL ;
   Spare02 : BOOL ;
  END_STRUCT ;
  intSavedPT : INT ;
END_VAR
VAR_TEMP
  tmpDeltaTime : INT ;
  tmpPulseIn : BOOL ;
END_VAR
BEGIN
NETWORK
TITLE = Inputs
      L     #PT;
      T     #CNT.PV;
// 
      A     #IN;
      FP    #EdgeIN;
      =     #tmpPulseIn;
      A     #IN;
      AN    #TON;	// [2.0]
      O;	// [2.0]
      AN    #IN;	// [2.0]
      A     #TON;	// [2.0]
      S     #CNT.LOAD;
// 
      A     #IN;	// [2.0]
      ON    #TON;	// [2.0]
      AN    #BREAK;
      A     "SYS_Scan0_Tick1s";
      AN    #CNT.QD;
      =     #CNT.CD;
NETWORK
TITLE = Handling of target time changes
      NOP   0;
//-Calculate time difference---
      L     #PT;
      L     #intSavedPT;
      -I;
      T     #tmpDeltaTime;
      JZ    NCHV;
// 
//-Restart the counter---
      A     #ParRestart;
      O     #CNT.LOAD;	// [2.0]
      JCN   RECA;
      S     #CNT.LOAD;
      JU    NCHV;
// 
//-Recalc the counter---
RECA: A     #ParRecalc;
      JCN   NRCA;
      L     #CNT.CV;
      L     #tmpDeltaTime;
      +I;
      JMZ   RERE;
      T     #CNT.PV;	// New value > 0
      S     #CNT.LOAD;
      JU    NCHV;
RERE: S     #CNT.R;	// New value <= 0
      JU    NCHV;
// 
//-Reload the counter---
NRCA: L     #CNT.CV;
      L     #CNT.PV;
      >I;
      JCN   NCHV;
      S     #CNT.LOAD;
      JU    NCHV;
// 
//-Save the new PT value---
NCHV: L     #PT;
      T     #intSavedPT;
NETWORK
TITLE = Call counter
      A     #IN;	//[2.0]
      ON    #TON;	//[2.0]
      AN    #CNT.QD;
      AN    #BREAK;
      A     "SYS_Scan0_Tick1s";
      JCN   ETn1;
      L     #ET;
      +     1;
      T     #ET;
ETn1: NOP   0;
// 
      CALL  #CNT;
      SET;
      R     #CNT.LOAD;
      R     #CNT.R;
// 
NETWORK
TITLE = Outputs
      L     #PT;
      T     #CNT.PV;	// Reload target value after recalculation
// 
      AN    #IN;	//[2.0]
      A     #TON;	//[2.0]
      O     #tmpPulseIn;
      AN    #Q;
      JCN   ETE;
      L     0;
      T     #ET;
ETE:  NOP   0;
// 
      L     #CNT.CV;
      T     #RT;
// 
      AN    #CNT.QD;
      AN    #TON;	// [2.0]
      O;	// [2.0]
      A     #CNT.QD;	// [2.0]
      A     #TON;	// [2.0]
      =     #Q;
NETWORK
TITLE = End of block
      BE;
END_FUNCTION_BLOCK

FUNCTION_BLOCK "STD_PULSEGEN"	// FB 1707
TITLE = Pulse generator with break possibility
//COPYRIGHT:    (C) 2004 BY  BUHLER LTD.
//                           CH-9240 UZWIL  SWITZERLAND
//
//PRODUCT:      STD_MU664    
//
//TITLE:        Pulse generator with break functionality
//              
//              Taktgenerator mit Unterbrechungsfunktionalität
//
//    
//
//--------------------------------------------------------------------------------
//
//IDENT:        AUTOR:              DEPT:                              DATE:
//STD_FB1707.1.0Ph. Engler          MU664                              22-Sep-2004
//              1st Release
//
//--------------------------------------------------------------------------------
//
//PURPOSE:      
//
//RESTRICTIONS:
//
//--------------------------------------------------------------------------------
//
AUTHOR : PE
FAMILY : STD
VERSION : 1.0
VAR_INPUT
  IN : BOOL ;
  BREAK : BOOL ;
  OnTime : INT ;
  OffTime : INT ;
END_VAR
VAR_OUTPUT
  Q : BOOL ;
  RTOn : INT ;
  RTOff : INT ;
END_VAR
VAR
  StaOnTime : BOOL ;
  EdgeOnTime : BOOL ;
  TON_OnTime : FB 1704;
  TON_OffTime : FB 1704;
END_VAR
BEGIN
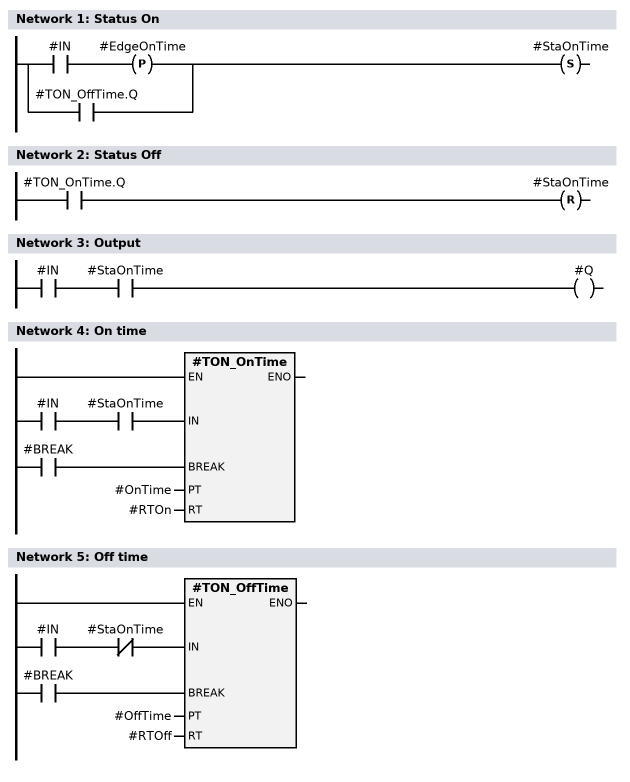
NETWORK
TITLE = Status On
      A     #IN;
      FP    #EdgeOnTime;
      O     #TON_OffTime.Q;
      S     #StaOnTime;
NETWORK
TITLE = Status Off
      A     #TON_OnTime.Q;
      R     #StaOnTime;
NETWORK
TITLE = Output
      A     #IN;
      A     #StaOnTime;
      =     #Q;
NETWORK
TITLE = On time
      A     #IN;
      A     #StaOnTime;
      =     L 0.0;
      BLD   103;
      A     #BREAK;
      =     L 0.1;
      BLD   103;
      CALL  #TON_OnTime (
           IN                       := L 0.0,
           BREAK                    := L 0.1,
           PT                       := #OnTime,
           RT                       := #RTOn);
      NOP   0;
NETWORK
TITLE = Off time
      A     #IN;
      AN    #StaOnTime;
      =     L 0.0;
      BLD   103;
      A     #BREAK;
      =     L 0.1;
      BLD   103;
      CALL  #TON_OffTime (
           IN                       := L 0.0,
           BREAK                    := L 0.1,
           PT                       := #OffTime,
           RT                       := #RTOff);
      NOP   0;
NETWORK
TITLE = End of block
END_FUNCTION_BLOCK

FUNCTION_BLOCK "STD_BranIntermitted"	// FB 1802
TITLE = STD: Intermitted mode of bransilos
//COPYRIGHT:    (C) 2004  BUHLER AG, CH-9240 UZWIL, SWITZERLAND
//
//PRODUCT:      STD_MU664
//
//TITLE:        Intermitted mode of bransilos
//
//              Intervallbetrieb von Kleiensilos
//
//
//--------------------------------------------------------------------------------
//
//IDENT:         AUTHOR:             DEPT:                             DATE:
//
//STD_FB1802.2.0 Ph. Engler          MU664                             06-Dec-2002
//               - InTick as Input for the time base
//               - OutRun to start external functions
//STD_FB1802.1.0 Ph. Engler          MU664                             07-Oct-2002
//               1st Release
//
//--------------------------------------------------------------------------------
//
//PURPOSE: 
//
//MANUAL : 
//
//RESTRICTIONS: 
//
//--------------------------------------------------------------------------------
//
AUTHOR : PE
FAMILY : STD
VERSION : 0.0
VAR_INPUT
  InTick : BOOL ;	//1Sek. = M 4.5; 1Min. = M 4.6
END_VAR
VAR
  StCode : INT ;	//State code
  InEnable : BOOL ;	//Release signal
  InDosing : BOOL ;	//Feedgroup of section is running
  StOff : BOOL ;	//Intermitted mode is off
  StRunning : BOOL ;	//Intermitted mode is on, the transport is running
  StPausing : BOOL ;	//Intermitted mode is on, the transport is stopped
  StWaiting : BOOL ;	//Intermitted mode is on, the feedgroups are stopped
  spare46 : BOOL ;
  spare47 : BOOL ;
  OutRun : BOOL ;	//Signal to start extern functions
  ParRunningTime : INT ;	//Running time in minutes
  ParPausingTime : INT ;	//Pausing time in minutes
  ActTime : INT ;	//Actual running or pausing time
  ActDiffTime : INT ;	//Actual rest time until timer elaps
  ActMaxTime : INT ;	//Actual target time
  CntCounter : SFB 2;	//Internal the timer is handled by a IEC-Counter
END_VAR
BEGIN
NETWORK
TITLE = States
      NOP   0;
//-StOff---
      A     #StOff;
      JC    StOf;
//-StRunning---
      A     #StRunning;
      JC    StRu;
//-StPausing---
      A     #StPausing;
      JC    StPa;
//-StWaiting---
      A     #StWaiting;
      JC    StWa;
//-Init---
      JU    StOf;
NETWORK
TITLE = StOff
StOf: SET;
      S     #StOff;
      S     #CntCounter.LOAD;
//-Transition to StRunning---
      A     #InEnable;
      R     #StOff;
      S     #StRunning;
      S     #CntCounter.R;
      JC    CC01;
// 
      JU    cnt;
NETWORK
TITLE = StRunning
StRu: SET;
      S     #StRunning;
// 
//-Counter target value---
      L     #ParRunningTime;
      L     32767;
      AW;
      T     #CntCounter.PV;
// 
//-Transition to StOff---
      AN    #InEnable;
      R     #StRunning;
      JC    StOf;
// 
//-Transition to StPausing---
      A     #CntCounter.QU;
      R     #StRunning;
      S     #StPausing;
      S     #CntCounter.R;
      JC    cnt;
// 
//-Transition to StWaiting---
      AN    #InDosing;
      R     #StRunning;
      JC    StWa;
// 
      JU    cnt;
NETWORK
TITLE = StPausing
StPa: SET;
      S     #StPausing;
// 
//-Counter target value---
      L     #ParPausingTime;
      L     32767;
      AW;
      T     #CntCounter.PV;
// 
//-Transition to StOff---
      AN    #InEnable;
      R     #StPausing;
      JC    StOf;
// 
//-Transition to StRunning---
      A     #CntCounter.QU;
      R     #StPausing;
      S     #StRunning;
      S     #CntCounter.R;
      JC    cnt;
// 
      JU    cnt;
NETWORK
TITLE = StWaiting
StWa: SET;
      S     #StWaiting;
// 
//-Transition to StOff---
      AN    #InEnable;
      R     #StWaiting;
      JC    StOf;
// 
//-Transition to StRunning---
      A     #InDosing;
      R     #StWaiting;
      JC    StRu;
// 
      JU    cnt;
NETWORK
TITLE = CU Count up
cnt:  A     #StRunning;
      A     #InDosing;
      O     #StPausing;
      A     #InTick;
      AN    #CntCounter.QU;
      =     #CntCounter.CU;
NETWORK
TITLE = CC Call counter
CC01: CALL  #CntCounter;
      SET;
      R     #CntCounter.R;
      R     #CntCounter.LOAD;
// 
NETWORK
TITLE = TV Time values
      NOP   0;
//-ActTime---
      L     #CntCounter.CV;
      T     #ActTime;
// 
//-ActDiffTime---
      L     #CntCounter.PV;
      L     #CntCounter.CV;
      -I;
      T     #ActDiffTime;
// 
//-ActMaxTime---
      L     #CntCounter.PV;
      T     #ActMaxTime;
NETWORK
TITLE = Outputs
      A     #StRunning;
      O     #StWaiting;
      =     #OutRun;
NETWORK
TITLE = State code
//State          StCode
// ---------------------
// StOff              1
// StRunning          2
// StPausing          3
// StWaiting          4
      AN    #StOff;
      JC    STC1;
      L     1;	// Code: StOff
      JU    STC9;
STC1: AN    #StRunning;
      JC    STC2;
      L     2;	// Code: StRunning
      JU    STC9;
STC2: AN    #StPausing;
      JC    STC3;
      L     3;	// Code: StPausing
STC3: AN    #StWaiting;
      JC    STC9;
      L     4;	// Code: StWaiting
STC9: T     #StCode;	// Old state code
NETWORK
TITLE = End of block
      BE;
END_FUNCTION_BLOCK

FUNCTION_BLOCK "STD_DryIntervalFilling"	// FB 1803
TITLE = STD: Intervall and dryfilling
//COPYRIGHT:    (C) 2000  BUHLER AG, CH-9240 UZWIL, SWITZERLAND
//
//PRODUCT:      STD_MU664
//
//TITLE:        Intervall and dryfilling of wheat bins
//
//              Intervall- und Trockenbefüllung von Weizenzellen
//
//
//--------------------------------------------------------------------------------
//
//IDENT:        AUTHOR:             DEPT:                              DATE:
//
//STD_FB1803.2.0 Ph. Engler          MU664                             11-Feb-2004
//               GCS7
//STD_FB1803.1.0 Ph. Engler          MU664                             07-Dec-2002
//               1st Release
//
//--------------------------------------------------------------------------------
//
//PURPOSE: 
//
//MANUAL : 
//
//RESTRICTIONS: 
//
//--------------------------------------------------------------------------------
//
AUTHOR : PE
FAMILY : STD
VERSION : 2.0
VAR_INPUT
  Code : INT ;
  RcvObject : BLOCK_DB ;
  InTick : BOOL ;	//1Sek. = M 4.5; 1Min. = M 4.6
END_VAR
VAR
  StCode : INT ;	//State code
  InIntervalFilling : BOOL ;	//Release signal for the intervall filling.
  InDryFilling : BOOL ;	//Release signal for the dry filling.
  InDosing : BOOL ;	//Feedgroup of section is running.
  InWaterRunning : BOOL ;	//Water valve is open.
  InEnable : BOOL ;	//Job is active.
  spare85 : BOOL ;
  spare86 : BOOL ;
  spare87 : BOOL ;
  StOff : BOOL ;
  StIntervalFilling : BOOL ;
  StDrying : BOOL ;
  StDryFilling : BOOL ;
  StWaiting : BOOL ;	//The feedgroups are stopped
  spare95 : BOOL ;
  spare96 : BOOL ;
  spare97 : BOOL ;
  OutNextReceiver : BOOL ;	//Signal to change the receiver
  OutEnableWater : BOOL ;	//Signal to start the water dosing
  OutDryFillingRequest : BOOL ;
  OutEdgeNextRcv : BOOL ;
  OutLoadedWet : BOOL ;	//Transfer machines are loaded with wet product.
  OutDryFillingDone : BOOL ;
  OutEdgeDryFillingTime : BOOL ;
  InDryFillingWeight : DINT ;
  ParDryFillingTime : BOOL ;	//Max. dryfilling time is active
  ParIntervalTime : INT ;	//Interval filling time
  ParMaxDryTime : INT ;	//Max. dry filling time
  ParDryingTime : INT ;	//Time to drying the transport elements
  ActTime : INT ;	//Actual running or pausing time
  ActDiffTime : INT ;	//Actual rest time until timer elaps
  ActMaxTime : INT ;	//Actual target time
  CntDryInterval1 : SFB 2;	//Internal the timer is handled by a IEC-Counter
  CntDrying : SFB 2;	//Time to drying the transport element after the dampener
  Bin : STRUCT
   BinNr : INT ;
   InfLevelWarning : BOOL ;
   InfLevelFault : BOOL ;
   OutDryFillingDone : BOOL ;
   user03 : BOOL ;
   VarFlagOverwriteLevel : BOOL ;
   InfLowLevel : BOOL ;
   InfLevelMiddle : BOOL ;
   InfHighLevel : BOOL ;
   InfActiveBin : BOOL ;
   InfPreselect : BOOL ;
   InfDeselect : BOOL ;
   StaEmpty : BOOL ;
   spare14 : BOOL ;
   spare15 : BOOL ;
   VarFlagLocked : BOOL ;
   VarFlagLevelFault : BOOL ;
   ParEmptyingTime : INT ;
   ActWeight : DINT ;
  END_STRUCT ;
END_VAR
VAR_TEMP
  VarAddrBin : DWORD ;
  VarAddrBinStatus : DWORD ;
  VarAddrActWeight : DWORD ;
  VarCnt : INT ;	//Loop counter
  VarDiNo : INT ;
  tmpDryFillingTimeOn : BOOL ;
END_VAR
BEGIN
NETWORK
TITLE = Open silo object db
      T     LD 17;
      TAK;
      T     LD 21;
      L     #RcvObject;
      T     LW 25;
      L     LD 21;
      L     LD 17;
      OPN   DB [LW 25];
NETWORK
TITLE = IN PLC new start or new binlist DB
      L     1;
      L     #Code;
      ==I;
      ON    DBX 63.6;	// InfInitDone
      JCN   IN00;
// 
      SET;
      S     DBX 63.6;	// --> InfInitDone
// 
      L     DBB 9;	// )  par_DW_first_bin
      SLD   3;	// )
      T     #VarAddrBin;	// --> Adresse first_bin
      L     0;	// ====START LOOP BIN ============
      L     DBB 13;	//  )  par_nr_of_bin
      ==I;
      BEC;
IN01: T     #VarCnt;
//-Load bin---
      L     P##Bin;
      T     #VarAddrBinStatus;
      L     DBD [#VarAddrBin];	//  )  Bin[x].BinNr / BinStatus
      T     DID [#VarAddrBinStatus];	//  )  BinStatus
//-Update StaEmpty--- 
      SET;
      =     #Bin.StaEmpty;
//-Save bin---
      L     DID [#VarAddrBinStatus];	//  )  BinStatus
      T     DBD [#VarAddrBin];	//  )  Bin[x].BinNr / BinStatus
      L     #VarAddrBin;
      L     DBB 11;	//  )  ParNrOfBytePerBin
      SLD   3;
      +D;	//  )
      T     #VarAddrBin;	//  )
//-Loop---
      L     #VarCnt;
      LOOP  IN01;	// ====END LOOP BIN ==============
// 
      BEU;
IN00: NOP   0;
NETWORK
TITLE = AS All states
      NOP   0;
//-LoadedWet---
      A     #InWaterRunning;
      S     #OutLoadedWet;
// 
//-Dry filling time switched on--- 
      A     #ParDryFillingTime;
      FP    #OutEdgeDryFillingTime;
      =     #tmpDryFillingTimeOn;
      A     #tmpDryFillingTimeOn;
      A     #StDryFilling;
      S     #CntDryInterval1.R;
// 
//-Dryfilling requested---
      CLR;
      =     #OutDryFillingRequest;
      =     #OutDryFillingDone;
// 
      L     DBB 9;	// )  par_DW_first_bin
      SLD   3;	// )
      T     #VarAddrBin;	// --> Adresse first_bin
      L     DBB 9;	// )  par_DW_first_bin
      L     6;
      +I;
      SLD   3;	// )
      T     #VarAddrActWeight;	// --> Adresse first actual weight
      L     0;	// ====START LOOP BIN ============
      L     DBB 13;	//  )  par_nr_of_bin
      ==I;
      BEC;
AS01: T     #VarCnt;
//-Load bin---
      L     P##Bin;
      T     #VarAddrBinStatus;
      L     DBD [#VarAddrBin];	//  )  Bin[x].BinNr / BinStatus
      T     DID [#VarAddrBinStatus];	//  )  BinStatus
//-OutDryFillingRequest--- 
      A     #Bin.InfActiveBin;
      O     #Bin.InfPreselect;
      A     #Bin.StaEmpty;
      A     #InDryFilling;
      S     #OutDryFillingRequest;
//-Update StaEmpty--- 
      A     #CntDryInterval1.QU;
      A     #StDryFilling;
      A     #ParDryFillingTime;
      AN    #tmpDryFillingTimeOn;
//      ON    #InDryFilling
      O(;
      L     DBD [#VarAddrActWeight];	//  )  Bin[x].BinNr / BinStatus
      L     #InDryFillingWeight;
      >=D;
      );
      A     #Bin.InfActiveBin;
      ON    #Bin.InfLowLevel;
      A     #InEnable;
      A     #Bin.StaEmpty;
      R     #Bin.StaEmpty;
//-OutDryFillingDone---
      S     #OutDryFillingDone;
//-Save bin---
      L     DID [#VarAddrBinStatus];	//  )  BinStatus
      T     DBD [#VarAddrBin];	//  )  Bin[x].BinNr / BinStatus
//-Next---
      L     #VarAddrBin;
      L     DBB 11;	//  )  ParNrOfBytePerBin
      SLD   3;
      +D;	//  )
      T     #VarAddrBin;	//  )
      L     #VarAddrActWeight;
      L     DBB 11;	//  )  ParNrOfBytePerBin
      SLD   3;
      +D;	//  )
      T     #VarAddrActWeight;	//  )
//-Loop---
      L     #VarCnt;
      LOOP  AS01;	// ====END LOOP BIN ==============
// 
//-Interval filling off---
      L     #ParIntervalTime;
      L     0;
      <=I;
      R     #InIntervalFilling;
// 
//-Dry filling off---
      L     #ParMaxDryTime;
      L     0;
      <=I;
      A     #ParDryFillingTime;
      R     #InDryFilling;
NETWORK
TITLE = States
      NOP   0;
//-StOff---
      A     #StOff;
      JC    StOf;
//-StIntervalFilling---
      A     #StIntervalFilling;
      JC    StIF;
//-StDrying---
      A     #StDrying;
      JC    StDR;
//-StDryFilling---
      A     #StDryFilling;
      JC    StDF;
//-StWaiting---
      A     #StWaiting;
      JC    StWa;
//-Init---
      JU    StOf;
NETWORK
TITLE = StOff
StOf: SET;
      S     #StOff;
      S     #CntDryInterval1.LOAD;
// 
//-Transition to StWaiting---
//      U     #InDryFilling
//      O     #InIntervalFilling
      A     #InEnable;
      R     #StOff;
      S     #StWaiting;
      S     #CntDryInterval1.R;
      S     #CntDrying.R;
      JC    CC01;
// 
      JU    cnt;
NETWORK
TITLE = StIntervalFilling
StIF: SET;
      S     #StIntervalFilling;
// 
//-Counter target value---
      L     #ParIntervalTime;
      L     32767;
      AW;
      T     #CntDryInterval1.PV;
// 
//-Transition to StOff---
      AN    #InIntervalFilling;
      AN    #InDryFilling;
      ON    #InEnable;
      R     #StIntervalFilling;
      JC    StOf;
// 
//-Transition to StDrying---
      A     #OutDryFillingRequest;
      A     #InDryFilling;
      A     #OutLoadedWet;
      R     #StIntervalFilling;
      S     #StDrying;
      S     #CntDrying.R;
      JC    cnt;
// 
//-Transition to StDryFilling---
      A     #OutDryFillingRequest;
      A     #InDryFilling;
      R     #StIntervalFilling;
      S     #StDryFilling;
      S     #CntDryInterval1.R;
      JC    cnt;
// 
//-Transition to StWaiting---
      AN    #InDosing;
      ON    #InIntervalFilling;
      R     #StIntervalFilling;
      S     #CntDrying.R;
      JC    StWa;
// 
      JU    cnt;
NETWORK
TITLE = StDrying
StDR: SET;
      S     #StDrying;
      S     #CntDryInterval1.LOAD;
// 
//-Transition to StOff---
      AN    #InIntervalFilling;
      AN    #InDryFilling;
      ON    #InEnable;
      R     #StDrying;
      JC    StOf;
// 
//-Transition to StIntervallFilling---
      AN    #OutDryFillingRequest;
      ON    #InDryFilling;
      R     #StDrying;
      S     #StIntervalFilling;
      S     #CntDryInterval1.R;
      JC    cnt;
// 
//-Transition to StDryFilling---
      A     #CntDrying.QU;
      R     #StDrying;
      S     #StDryFilling;
      R     #OutLoadedWet;
      S     #CntDryInterval1.R;
      JC    cnt;
// 
      JU    cnt;
NETWORK
TITLE = StDryFilling
StDF: SET;
      S     #StDryFilling;
      AN    #ParDryFillingTime;
      S     #CntDryInterval1.LOAD;
// 
//-Counter target value---
      L     #ParMaxDryTime;
      L     32767;
      AW;
      T     #CntDryInterval1.PV;
// 
//-Transition to StOff---
      AN    #InIntervalFilling;
      AN    #InDryFilling;
      ON    #InEnable;
      R     #StDryFilling;
      JC    StOf;
// 
//-Transition to StIntervallFilling---
      AN    #OutDryFillingRequest;
      ON    #InDryFilling;
      R     #StDryFilling;
      S     #StIntervalFilling;
      S     #CntDryInterval1.R;
      JC    cnt;
// 
//-Transition to StWaiting---
      AN    #InDosing;
      R     #StDryFilling;
      JC    StWa;
// 
      JU    cnt;
NETWORK
TITLE = StWaiting
StWa: SET;
      S     #StWaiting;
      AN    #OutDryFillingRequest;
      ON    #ParDryFillingTime;
      AN    #InIntervalFilling;
      S     #CntDryInterval1.LOAD;
// 
//-Transition to StOff---
//      UN    #InIntervalFilling
//      UN    #InDryFilling
      ON    #InEnable;
      R     #StWaiting;
      JC    StOf;
// 
//-Transition to StIntervallFilling---
      A     #InDosing;
      A     #InIntervalFilling;
      AN    #OutDryFillingRequest;
      R     #StWaiting;
      AN    #StWaiting;
      A     #CntDryInterval1.QU;
      S     #CntDryInterval1.R;
      AN    #StWaiting;
      JC    StIF;
// 
//-Transition to StDrying---
      A     #InDosing;
      A     #OutDryFillingRequest;
      AN    #CntDrying.QU;
      R     #StWaiting;
      JC    StDR;
// 
//-Transition to StDryFilling---
      A     #InDosing;
      A     #OutDryFillingRequest;
      R     #StWaiting;
      JC    StDF;
// 
      JU    cnt;
NETWORK
TITLE = DT Drying Time
cnt:  A     #StDrying;
      A     #InTick;
      AN    #CntDrying.QU;
      =     #CntDrying.CU;
// 
//-Counter target value---
      L     #ParDryingTime;
      L     32767;
      AW;
      T     #CntDrying.PV;
// 
//-Counter dry filling--- 
      CALL  #CntDrying;
      SET;
      R     #CntDrying.R;
      R     #CntDrying.LOAD;
// 
NETWORK
TITLE = Interval and dry filling time
      A     #StDryFilling;
      A     #ParDryFillingTime;
      O     #StIntervalFilling;
      T     LD 17;
//      U     DBX   43.4                  // .ToASW.InfWayAdjustEnd
      TAK;	// .ToASW.InfPreselect
      T     LD 21;
      L     #RcvObject;
      T     LW 25;
// 
      L     LD 21;
      L     LD 17;	// .ToASW.InfPreselect
      OPN   DB [LW 25];
      AN    DBX 43.1;
// 
      A     #InTick;
      AN    #CntDryInterval1.QU;
      =     #CntDryInterval1.CU;
      T     LD 17;
      TAK;
      T     LD 21;
      L     #RcvObject;
      T     LW 25;
      L     LD 21;
// 
      L     LD 17;
      OPN   DB [LW 25];
      A     DBX 43.1;
      AN    #StDrying;
      S     #CntDryInterval1.R;
CC01: CALL  #CntDryInterval1;
      SET;
      R     #CntDryInterval1.R;
      R     #CntDryInterval1.LOAD;
NETWORK
TITLE = TV Time values
      NOP   0;
//-ActTime---
      L     #CntDryInterval1.CV;
      T     #ActTime;
// 
//-ActDiffTime---
      L     #CntDryInterval1.PV;
      L     #CntDryInterval1.CV;
      -I;
      T     #ActDiffTime;
// 
//-ActMaxTime---
      L     #CntDryInterval1.PV;
      T     #ActMaxTime;
NETWORK
TITLE = Outputs
      NOP   0;
//-OutEnableWater---
      A     #StOff;
      O     #StIntervalFilling;
      O(;
      AN    #InDryFilling;
      ON    #OutDryFillingRequest;
      A     #StWaiting;
      );
      =     #OutEnableWater;
// 
//-OutNextReceiver---
      A     #StIntervalFilling;
      A     #CntDryInterval1.QU;
      O     #OutDryFillingDone;
      FP    #OutEdgeNextRcv;
      T     LD 17;
      TAK;	// .ToSSW.CmdNext
      T     LD 21;
      L     #RcvObject;
      T     LW 25;
      L     LD 21;
      L     LD 17;
      OPN   DB [LW 25];
      S     DBX 62.6;
      S     #CntDryInterval1.R;
NETWORK
TITLE = State code
//State          StCode
// ---------------------
// StOff              1
// StIntervalFilling  2
// StDrying           3
// StDryFilling       4
// StWaiting          5
// StUpToHL           6
      L     1;
      A     #StOff;
      JC    STCS;
      L     2;
      A     #StIntervalFilling;
      JC    STCS;
      L     3;
      A     #StDrying;
      JC    STCS;
      L     4;
      A     #StDryFilling;
      JC    STCS;
      L     6;
      A     #InDryFilling;
      AN    #OutDryFillingRequest;
      AN    #InIntervalFilling;
      O(;
      AN    #InIntervalFilling;
      AN    #InDryFilling;
      );
      A     #StWaiting;
      JC    STCS;
      L     5;
      A     #StWaiting;
      JC    STCS;
      L     0;	// Default value
STCS: T     #StCode;
NETWORK
TITLE = End of block
      BE;
END_FUNCTION_BLOCK

